# B&R Automation Studio project baseProject
Automation Studio 6.3.1.32; technology packages: mappCockpit 6.2.1, mappMotion 6.3.1, mappSafety 6.2.0, mappServices 6.3.3, mappView 6.3.1, OpcUaCs 6.0.0

## Configuration Config1

CPU X20CP1684, AutomationRuntime 6.0.2, Build 11.3.0, Vc 6.0.0

### Task classes (Cpu.sw)
```
Cyclic#4 (cycle 16000 us, tolerance 16000 us):
  HMI <- HMI.prg
  Safety <- Safety.prg
  motion <- motion.prg
  mappIO <- mappIO.prg
  mappAlarmX <- mappAlarmX.prg
  mappRecipe <- mappRecipe.prg
  EventLog <- EventLog.prg
  Robot <- Robot.prg
Libraries: AsIOAcc, runtime, AsZip, FileIO, astime, sys_lib, ArEventLog, AsBrStr, CoTrace, SfDomain, DataObj, AsMem, AsArProf, standard, MpAlarmX, MpBase, MpAxis, McBase, MpSequence, MpAudit, MpRecipe, MpUserX, MpReport, MpSkyline, MpFile, MpPackML, MpCodeBox, MpCom, MpIO, McAxis, McAcpAx, MpServer
```

### Hardware
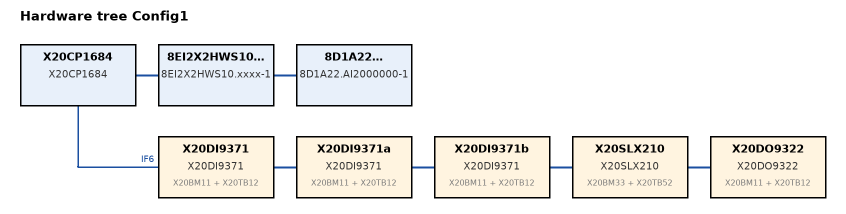
```
8D1A22.AI2000000-1 : 8D1A22.AI2000000-1 v1.0.1.0 (NodeNumber=2)  [PLK1 -> 8EI2X2HWS10.xxxx-1.PLK2 [Cable Type=PowerlinkCable, Length=10, Version=1.0.0.3]]
8EI2X2HWS10.xxxx-1 : 8EI2X2HWS10.xxxx-1 v2.4.0.0 (NodeNumber=1)  [PLK1 -> X20CP1684.IF3 [Cable Type=PowerlinkCable, Length=10, Version=1.0.0.3]; PLK2 -> 8D1A22.AI2000000-1.PLK1 [Cable Type=PowerlinkCable, Length=10, Version=1.0.0.3]]
  DriveConfiguration/Module:
    McAcoposTypeID = AcoposP3SConfig
    ActivateACOPOSSimulationOnPLC = 1
    PowerSupply = AC
  DriveConfiguration/Encoder/EncoderX41:
    InterfaceType = NotUsed
  DriveConfiguration/Channel[1]/RealAxis:
    AxisReference = gAxis_1
    MechanicalElementsIsInvisible = 0
  DriveConfiguration/Channel[1]/RealAxis/MechanicalElements/Gearbox:
    InputIsReadOnly = 0
    Input = 1
    OutputIsReadOnly = 0
    Output = 1
  DriveConfiguration/Channel[1]/RealAxis/MechanicalElements/RotaryToLinearTransformation:
    ReferenceDistanceIsReadOnly = 0
    ReferenceDistance = 1
  DriveConfiguration/Channel[1]/RealAxis:
    EncoderLink = OneEncoder
  DriveConfiguration/Channel[1]/RealAxis/Controller:
    ModeIsReadOnly = 0
    Mode = PositionController
  DriveConfiguration/Channel[1]/RealAxis/Homing:
    ModeIsReadOnly = 0
    Mode = Direct
    RestorePositionVariable = 
  DriveConfiguration/Channel[1]/RealAxis/StopReaction:
    QuickstopIsReadOnly = 0
    Quickstop = DecelerationLimit
    DriveErrorIsReadOnly = 0
    DriveError = DecelerationLimit
  DriveConfiguration/Channel[1]/RealAxis/MovementErrorLimits:
    PositionError = 10.0
    VelocityErrorMonitoring = Automatic1
  DriveConfiguration/Channel[1]/RealAxis:
    JerkFilterIsReadOnly = 0
    JerkFilter = NotUsed
    ZeroVibrationFilter = NotUsed
  DriveConfiguration/Channel[1]/RealAxis/DigitalInputs/HomingSwitch:
    SourceIsReadOnly = 0
    Source = NotUsed
    Level = High
  DriveConfiguration/Channel[1]/RealAxis/DigitalInputs/PositiveLimitSwitch:
    SourceIsReadOnly = 0
    Source = NotUsed
    Level = High
  DriveConfiguration/Channel[1]/RealAxis/DigitalInputs/NegativeLimitSwitch:
    SourceIsReadOnly = 0
    Source = NotUsed
    Level = High
  DriveConfiguration/Channel[1]/RealAxis/DigitalInputs/Trigger1:
    Source = X8Trigger1
    Level = High
  DriveConfiguration/Channel[1]/RealAxis/DigitalInputs/Trigger2:
    Source = X8Trigger2
    Level = High
  DriveConfiguration/Channel[1]/RealAxis/DigitalInputs/Quickstop:
    Input = Trigger2
  DriveConfiguration/Channel[1]/RealAxis/Simulation:
    SimulationModeOnPLC = SetValueGeneration
    SimulationModeOnACOPOS = NotUsed
  DriveConfiguration/Channel[1]:
    VirtualAxis = NotUsed
    ExternalEncoderAxis = NotUsed
X20BM11 : X20BM11 v1.1.0.0  [X2X1 -> X20CP1684.IF6]
X20BM11a : X20BM11 v1.1.0.0  [X2X1 -> X20BM11b.X2X2]
X20BM11b : X20BM11 v1.1.0.0  [X2X1 -> X20BM11.X2X2]
X20BM11c : X20BM11 v1.1.0.0  [X2X1 -> X20BM33.X2X2]
X20BM33 : X20BM33 v1.1.0.0  [X2X1 -> X20BM11a.X2X2]
X20CP1684 : X20CP1684 v1.8.1.0
  Connector IF2:
    ActivateDevice = 1
    Mode = Manual
    InternetAddress = 192.168.50.160
    SubnetMask = 255.255.255.0
  Connector IF3:
    CycleTime = 800
  ConfigurationID = mappView_Config1
  Simulation = 1
  TimerDeviceType = EPLX2X
  TimerDevice = X20CP1684.IF3
  IdleTaskClass = 8
  TaskClassIdleTime = 1600
  Cyclic1Duration = 800
  Cyclic1Tolerance = 0
  Cyclic2Duration = 1600
  Cyclic2Tolerance = 1600
  Cyclic3Duration = 6400
  Cyclic3Tolerance = 6400
  Cyclic4Duration = 16000
  Cyclic4Tolerance = 16000
  Cyclic8Duration = 9600
  FileDevice1
  FileDeviceName1 = USER
  FileDevicePath1 = USER_PATH
  FileDevice2
  FileDeviceName2 = CF
  FileDevicePath2 = C:\
  ActivateFtpServer = 1
  FTPProtocol = 1
  FtpUser1
  FtpUsername1 = ged
  FtpUserPassword1 = mhumPqqez6h0Xcak9Se1xIrLnNOPX6JLQ7ADh5QSq84=
  FtpUserSalt1 = ifft5IbT
  FTPAccessRight1 = 0
  ActivateWebServer = 1
  ActivateSdm = 1
X20DI9371 : X20DI9371 v1.6.1.0  [SS1 -> X20TB12.SS; SL -> X20BM11.SL1]
  Supervision = off
X20DI9371a : X20DI9371 v1.6.1.0  [SS1 -> X20TB12b.SS; SL -> X20BM11b.SL1]
  Supervision = off
X20DI9371b : X20DI9371 v1.6.1.0  [SS1 -> X20TB12a.SS; SL -> X20BM11a.SL1]
  Supervision = off
X20DO9322 : X20DO9322 v1.7.0.0  [SS1 -> X20TB12c.SS; SL -> X20BM11c.SL1]
  Supervision = off
X20SLX210 : X20SLX210 v2.6.1.0  [SS1 -> X20TB52.SS; SL -> X20BM33.SL1]
  Supervision = off
X20TB12 : X20TB12 v1.0.0.0
X20TB12a : X20TB12 v1.0.0.0
X20TB12b : X20TB12 v1.0.0.0
X20TB12c : X20TB12 v1.0.0.0
X20TB52 : X20TB52 v1.0.0.2
```

### IoMap.iom - X20CP1684/IoMap.iom
```iecst
VAR_CONFIG
	::doTestOutput01 AT %QX."X20DO9322".DigitalOutput01;
	::diTestInput01 AT %IX."X20DI9371".DigitalInput01;
	::diTestInput02 AT %IX."X20DI9371a".DigitalInput01;
END_VAR
```

### Config_1.axis - X20CP1684/mappMotion/Config_1.axis
```
Element gAxis_1 (Type=axis)
  BaseType = RotaryPeriodic
  MovementLimits = Internal
  Alarms = None
```

- Safety project (password-protected, skipped)

### Config_2.mpio - X20CP1684/mappServices/Config_2.mpio
```
Element gIoConfig (Type=mpio)
  mapp.Gen:
    Enable = TRUE
    EnableCockpit = TRUE
    Audit = TRUE
    Parent
  Import:
    Main = no
    ImportAllow
    AutoRestore = TRUE
    PreservePv = TRUE
    RemoveLinks = FALSE
    BackupLoc = USER
    TemplateLoc = USER
    Plausibility:
      AllowNarrow = FALSE
      CheckTypes = TRUE
      CheckPv = TRUE
      CheckAxPv = TRUE
  IoDatapoints:
    Inputs:
      0 = #global
    Outputs:
      0 = #global
  Alarms = MpAlarmX
    mapp.AlarmX.Core.Configuration:
      [0]:
        Name = ImportFailed
        Message = {$BR/mapp/MpIO/Alarms/ImportFailed}
        Code = 0
        Severity = 1
        Behavior = EdgeAlarm
          AutoReset = TRUE
          Acknowledge = 1
          Confirm = 0
          MultipleInstances = TRUE
          ReactionWhilePending = TRUE
          Async = FALSE
          Recording:
            InactiveToActive = TRUE
            ActiveToInactive = FALSE
            UnacknowledgedToAcknowledged = TRUE
            UnconfirmedToConfirmed = TRUE
        Disable = FALSE
        AdditionalInformation1
        AdditionalInformation2
      [1]:
        Name = ImportDone
        Message = {$BR/mapp/MpIO/Alarms/ImportDone}
        Code = 0
        Severity = 1
        Behavior = EdgeAlarm
          AutoReset = TRUE
          Acknowledge = 1
          Confirm = 0
          MultipleInstances = TRUE
          ReactionWhilePending = TRUE
          Async = FALSE
          Recording:
            InactiveToActive = TRUE
            ActiveToInactive = FALSE
            UnacknowledgedToAcknowledged = TRUE
            UnconfirmedToConfirmed = TRUE
        Disable = FALSE
        AdditionalInformation1
        AdditionalInformation2
      [2]:
        Name = HwChanged
        Message = {$BR/mapp/MpIO/Alarms/HwChanged}
        Code = 0
        Severity = 1
        Behavior = EdgeAlarm
          AutoReset = TRUE
          Acknowledge = 1
          Confirm = 0
          MultipleInstances = TRUE
          ReactionWhilePending = TRUE
          Async = FALSE
          Recording:
            InactiveToActive = TRUE
            ActiveToInactive = FALSE
            UnacknowledgedToAcknowledged = TRUE
            UnconfirmedToConfirmed = TRUE
        Disable = FALSE
        AdditionalInformation1
        AdditionalInformation2
```

### Config_4.mpalarmxlist - X20CP1684/mappServices/Config_4.mpalarmxlist
```
Element gAlarmXList (Type=mpalarmxlist)
  mapp.AlarmX.Core.Configuration:
    [0]:
      Name = TemperatureHigh
      Message = The Temperature is Too High
      Code = 100
      Severity = 10
      Behavior = PersistentAlarm
        Confirm = 0
        ReactionWhilePending = TRUE
        Retain = FALSE
        Async = FALSE
        DataUpdate:
          Activation:
            TimeStamp = FALSE
            Snippets = FALSE
        Recording:
          InactiveToActive = TRUE
          UnacknowledgedToAcknowledged = TRUE
          AcknowledgedToUnacknowledged = FALSE
          UnconfirmedToConfirmed = TRUE
          ConfirmedToUnconfirmed = FALSE
          Update = FALSE
      Disable = FALSE
      InhibitPV
      AdditionalInformation1
      AdditionalInformation2
  mapp.AlarmX.Snippets:
    AutoDetect = 1
      Language
```

### Config_7.mpfilemanager - X20CP1684/mappServices/Config_7.mpfilemanager
```
Element FileManagement (Type=mpfilemanager)
  mapp.Gen:
    Enable = TRUE
    EnableCockpit = TRUE
    Audit = TRUE
    Parent
  FileManager:
    USB = 1
    Devices:
      0:
        DeviceName = USER
        Text = User
    Access:
      0:
        Folder = *
        Roles:
          0:
            Role = Everyone
            Rights:
              Visible = TRUE
              FolderRead = TRUE
              FileRead = TRUE
              FileEdit = TRUE
              FolderEdit = TRUE
```

## Configuration mappDemoDefault

CPU X20CP1686X, AutomationRuntime 6.0.2, Build 11.3.0, Vc 

### Task classes (Cpu.sw)
```
Cyclic#1:
  MainContro <- MainControl.prg
  ConveyorSi <- ConveyorSim.prg
  Alarm <- Infrastructure.Alarm.prg
Cyclic#4:
  Recipe <- Infrastructure.Recipe.prg
  File <- Infrastructure.File.prg
  Audit <- Infrastructure.Audit.prg
  Report <- Infrastructure.Report.prg
  IO <- Infrastructure.IO.prg
  Sequence <- Infrastructure.Sequence.prg
  CodeBox <- Infrastructure.CodeBox.prg
  PackML <- Industry.PackML.prg
Cyclic#8:
  Skyline <- Infrastructure.Skyline.prg
Binaries: mvLoader, arsvcreg, TCLang, FWRules, udbdef, TCData, mvConfig, CfgFileUI, arconfig, UaCsConfig, CfgFile, mCoWebSc, CfgSkyline, User, TC, asfw, CfgAudit, iomap, Role, CfgReportF, CfgUserX, ashwd, CfgRecipe, CfgSeq, CfgReport, CfgComUnit, ashwac, sysconf, CfgCodeCor, Settings, CfgCodeBox, CfgIO, CfgPack, CfgAlaList, CfgAlaHist, CfgAlaCore, BRRole, CfgHistory, UaDvConfig, CfgAlarm
Libraries: Runtime, Operator, AsIecCon, astime, AsArSdm, DataObj, FileIO, AsBrStr, sys_lib, brsystem, AsArProf, AsMem, standard, AsBrWStr, ArTextSys, ArCert, ArSsl, AsETH, AsHW, AsIOMMan, AsUSB, AsZip, ArUser, UaCoal, UaCoalPrv, ArProject, AsARCfg, CoTrace, MpAlarmX, MpBase, MpSequence, MpAudit, MpRecipe, MpUserX, MpReport, MpSkyline, MpFile, MpPackML, MpCodeBox, MpCom, MpIO, MpServer
```

### Hardware
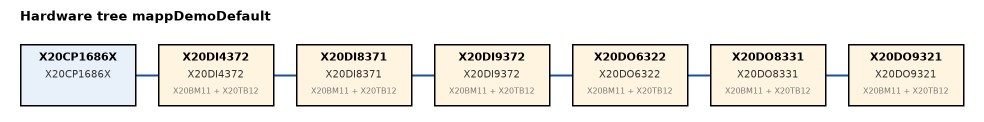
```
X20BM11 : X20BM11 v1.1.0.0  [X2X1 -> X20CP1686X.IF6]
X20BM11a : X20BM11 v1.1.0.0  [X2X1 -> X20BM11.X2X2]
X20BM11b : X20BM11 v1.1.0.0  [X2X1 -> X20BM11a.X2X2]
X20BM11c : X20BM11 v1.1.0.0  [X2X1 -> X20BM11b.X2X2]
X20BM11d : X20BM11 v1.1.0.0  [X2X1 -> X20BM11c.X2X2]
X20BM11e : X20BM11 v1.1.0.0  [X2X1 -> X20BM11d.X2X2]
X20CP1686X : X20CP1686X v1.8.2.0
  Connector IF2:
    ActivateDevice = 1
  ConfigurationID = mappServicesHighlights_Config1
  AutomaticTransferOfUserfiles = on
  Simulation = 1
  FileDevice1
  FileDeviceName1 = HD
  FileDevicePath1 = USER_PATH
  FileDevice2
  FileDeviceName2 = mappDir
  FileDevicePath2 = USER_PATH\mappDemo
  FileDevice3
  FileDeviceName3 = mappReport
  FileDevicePath3 = USER_PATH\mappDemo\Reports
  FileDevice4
  FileDeviceName4 = mappIO
  FileDevicePath4 = USER_PATH\IO
  FileDevice5
  FileDeviceName5 = mappIOBackup
  FileDevicePath5 = USER_PATH\IO\Backup
  FileDevice6
  FileDeviceName6 = mappSequence
  FileDevicePath6 = USER_PATH\Sequence
  FileDevice7
  FileDeviceName7 = mappCodeBox
  FileDevicePath7 = USER_PATH\CodeBox
  ActivateWebServer = 1
  WebServerProtocol = 1
  ActivateSdm = 1
X20DI4372 : X20DI4372 v1.4.1.0  [SS1 -> X20TB12.SS; SL -> X20BM11.SL1]
X20DI8371 : X20DI8371 v1.6.1.0  [SS1 -> X20TB12a.SS; SL -> X20BM11a.SL1]
X20DI9372 : X20DI9372 v1.6.1.0  [SS1 -> X20TB12b.SS; SL -> X20BM11b.SL1]
X20DO6322 : X20DO6322 v1.4.1.0  [SS1 -> X20TB12c.SS; SL -> X20BM11c.SL1]
X20DO8331 : X20DO8331 v1.2.2.0  [SS1 -> X20TB12d.SS; SL -> X20BM11d.SL1]
X20DO9321 : X20DO9321 v1.2.2.0  [SS1 -> X20TB12e.SS; SL -> X20BM11e.SL1]
X20TB12 : X20TB12 v1.0.0.0
X20TB12a : X20TB12 v1.0.0.0
X20TB12b : X20TB12 v1.0.0.0
X20TB12c : X20TB12 v1.0.0.0
X20TB12d : X20TB12 v1.0.0.0
X20TB12e : X20TB12 v1.0.0.0
```

### BRRole.brrole - X20CP1686X/AccessAndSecurity/UserRoleSystem/BRRole.brrole
```
Element BR_Anonymous (Type=BRRole)
Element BR_Engineer (Type=BRRole)
Element BR_Observer (Type=BRRole)
Element BR_SafetyAdmin (Type=BRRole)
Element BR_SecurityAdmin (Type=BRRole)
```

### CfgAlaCore.mpalarmxcore - X20CP1686X/mappServices/CfgAlaCore.mpalarmxcore
```
Element gAlarmXCore (Type=mpalarmxcore)
  mapp.Gen:
    Enable = TRUE
    TaskClass = 4
  mapp.AlarmX.List:
    [0]:
      List = gAlarmXCore_List
      Offset = 0
  mapp.AlarmX.Create = Disabled
  mapp.AlarmX.Core.Retain:
    Memory = 0
```

### CfgAlaHist.mpalarmxhistory - X20CP1686X/mappServices/CfgAlaHist.mpalarmxhistory
```
Element gAlarmXHistory (Type=mpalarmxhistory)
  mapp.Gen:
    Audit = TRUE
  mapp.AlarmX.History
```

### CfgAlaList.mpalarmxlist - X20CP1686X/mappServices/CfgAlaList.mpalarmxlist
```
Element gAlarmXCore_List (Type=mpalarmxlist)
  mapp.AlarmX.Core.Configuration:
    [0]:
      Name = RecordingStarted
      Message = {$mappDemo/MpDataUserAlarm}
      Code = 2501
      Behavior = UserDefined
        AutoReset = TRUE
        Acknowledge = 0
        Recording:
          ActiveToInactive = FALSE
    [1]:
      Name = WaterEmpty
      Message = {$IAT/AlarmWater}
      Code = 2503
      Behavior = LevelMonitoring
        Monitoring:
          MonitoredPV = ::MainContro:Refill[3]
          LowLimitEnable = Static
            Limit = 15
      AdditionalInformation1 = WaterEmpty
    [2]:
      Name = CoffeeEmpty
      Message = {$IAT/AlarmCoffee}
      Code = 2504
      Behavior = LevelMonitoring
        Monitoring:
          MonitoredPV = ::MainContro:Refill[0]
          LowLimitEnable = Static
            Limit = 15
      AdditionalInformation1 = CoffeeEmpty
    [3]:
      Name = MilkEmpty
      Message = {$IAT/AlarmMilk}
      Code = 2505
      Behavior = LevelMonitoring
        Monitoring:
          MonitoredPV = ::MainContro:Refill[1]
          LowLimitEnable = Static
            Limit = 15
      AdditionalInformation1 = MilkEmpty
    [4]:
      Name = SugarEmpty
      Message = {$IAT/AlarmSugar}
      Code = 2506
      Behavior = LevelMonitoring
        Monitoring:
          MonitoredPV = ::MainContro:Refill[2]
          LowLimitEnable = Static
            Limit = 15
      AdditionalInformation1 = SugarEmpty
    [5]:
      Name = ModuleAlarm
      Message = {$IAT/AlarmModule}
      Behavior = PersistentAlarm
  mapp.AlarmX.Snippets:
    [0]:
      Key = WaterLevel
      Value:
        PV = ::MainContro:Refill[3]
    [1]:
      Key = SugarLevel
      Value:
        PV = ::MainContro:Refill[2]
    [2]:
      Key = CoffeeLevel
      Value:
        PV = ::MainContro:Refill[0]
    [3]:
      Key = MilkLevel
      Value:
        PV = ::MainContro:Refill[1]
```

### CfgAudit.mpaudittrail - X20CP1686X/mappServices/CfgAudit.mpaudittrail
```
Element gAuditTrail (Type=mpaudittrail)
  mapp.Gen:
    Enable = TRUE
    TaskClass = 8
  Audit:
    Events:
      [0] = 600
      [1] = 400
      [2] = 1000
      [3] = 1001
      [4] = 1002
      [5] = 1003
      [6] = 700
      [7] = 701
      [8] = 702
      [9] = 703
      [10] = 704
      [11] = 100
      [12] = 101
      [13] = 102
      [14] = 103
      [15] = 104
      [16] = 105
      [17] = 106
      [18] = 107
      [19] = 108
      [20] = 150
      [21] = 151
      [22] = 152
      [23] = 153
      [24] = 154
      [25] = 155
      [26] = 156
      [27] = 157
      [28] = 158
      [29] = 159
      [30] = 160
      [31] = 161
      [32] = 162
      [33] = 163
      [34] = 164
      [35] = 165
      [36] = 166
      [37] = 167
      [38] = 168
      [39] = 169
      [40] = 170
      [41] = 171
      [42] = 300
      [43] = 301
      [44] = 302
      [45] = 303
      [46] = 350
      [47] = 351
      [48] = 352
      [49] = 353
    RecordMemory = 1
    RecordingSize = 200
    SramBufferSize = 4
    TextSource:
      DisplayFormat = {$AuditDisplay/Root}
      ExportFormat = {$AuditExport/Root}
    Archive = On
      Mode = 0
      Time = 0
      MaxSize = 100
    Export:
      RawData = FALSE
      FileType = 0
      Encrypt = FALSE
      PassPhrase = Insert your passphrase here...
  Monitor:
    0:
      pv = ::Recipe:CoffeeIngredients.Milk
      id = Milk
    1:
      pv = ::Recipe:CoffeeIngredients.Water
      id = Water
    2:
      pv = ::Recipe:CoffeeIngredients.Sugar
      id = Sugar
    3:
      pv = ::Recipe:CoffeeIngredients.Coffee
      id = Coffee
  Alarms = MpAlarmX
    mapp.AlarmX.Core.Configuration:
      [0]:
        Name = ArchiveAvailable
        Message = {$BR/mapp/MpAuditTrail/Alarms/ArchiveAvailable}
        Code = 0
        Severity = 1
        Behavior = PersistentAlarm
          AutoReset = FALSE
          Acknowledge = 1
          Confirm = 0
          MultipleInstances = FALSE
          ReactionWhilePending = TRUE
          Async = FALSE
          DataUpdate:
            Activation:
              TimeStamp = FALSE
              Snippets = FALSE
          Recording:
            InactiveToActive = TRUE
            ActiveToInactive = FALSE
            UnacknowledgedToAcknowledged = TRUE
            AcknowledgedToUnacknowledged = TRUE
            UnconfirmedToConfirmed = TRUE
            ConfirmedToUnconfirmed = TRUE
            Update = FALSE
        Disable = FALSE
        AdditionalInformation1
        AdditionalInformation2
      [1]:
        Name = MaxArchives
        Message = {$BR/mapp/MpAuditTrail/Alarms/MaxArchives}
        Code = 0
        Severity = 1
        Behavior = EdgeAlarm
          AutoReset = TRUE
          Acknowledge = 1
          Confirm = 0
          MultipleInstances = TRUE
          ReactionWhilePending = TRUE
          Async = FALSE
          Recording:
            InactiveToActive = TRUE
            ActiveToInactive = FALSE
            UnacknowledgedToAcknowledged = TRUE
            UnconfirmedToConfirmed = TRUE
        Disable = FALSE
        AdditionalInformation1
        AdditionalInformation2
```

### CfgComUnit.mpcomunit - X20CP1686X/mappServices/CfgComUnit.mpcomunit
```
Element gGroup (Type=mpcomunit)
  Display:
    Groups:
      0:
        Id = Fluid
        DisplayUnits:
          Metric:
            Code = MLT
          Imperial:
            Code = OZA
          ImperialUS:
            Code = OZA
      1:
        Id = Gram
        DisplayUnits:
          Metric:
            Code = GRM
          Imperial:
            Code = ONZ
          ImperialUS:
            Code = ONZ
    Datapoints:
      0:
        Id = ::Recipe:CoffeeIngredients.Milk
        DisplayUnits = UnitGroup
          Unitgroup = Fluid
      1:
        Id = ::Recipe:CoffeeIngredients.Water
        DisplayUnits = UnitGroup
          Unitgroup = Fluid
      2:
        Id = ::Recipe:CoffeeIngredients.Sugar
        DisplayUnits = UnitGroup
          Unitgroup = Gram
      3:
        Id = ::Recipe:CoffeeIngredients.Coffee
        DisplayUnits = UnitGroup
          Unitgroup = Gram
      4:
        Id = ::MainContro:Refill[1]
        DisplayUnits = UnitGroup
          Unitgroup = Fluid
      5:
        Id = ::MainContro:Refill[2]
        DisplayUnits = UnitGroup
          Unitgroup = Gram
      6:
        Id = ::MainContro:Refill[0]
        DisplayUnits = UnitGroup
          Unitgroup = Gram
      7:
        Id = ::MainContro:Refill[3]
        DisplayUnits = UnitGroup
          Unitgroup = Fluid
    Units:
      0:
        EngineeringUnit:
          Code = MLT
        DisplayUnits:
          Metric:
            Code = MLT
          Imperial:
            Code = MLT
          ImperialUS:
            Code = MLT
      1:
        EngineeringUnit:
          Code = MLT
        DisplayUnits:
          Metric:
            Code = MLT
          Imperial:
            Code = MLT
          ImperialUS:
            Code = MLT
      2:
        EngineeringUnit:
          Code = GRM
        DisplayUnits:
          Metric:
            Code = GRM
          Imperial:
            Code = ONZ
          ImperialUS:
            Code = ONZ
      3:
        EngineeringUnit:
          Code = GRM
        DisplayUnits:
          Metric:
            Code = GRM
          Imperial:
            Code = ONZ
          ImperialUS:
            Code = ONZ
```

### CfgFile.mpfilemanager - X20CP1686X/mappServices/CfgFile.mpfilemanager
```
Element FileManagement (Type=mpfilemanager)
  mapp.Gen:
    Enable = TRUE
    EnableCockpit = TRUE
    Audit = TRUE
    Parent
  FileManager:
    USB = 0
    Devices:
      0:
        DeviceName = mappDir
        Text = Recipe files
    Access:
      0:
        Folder = *
        Roles:
          0:
            Role = Everyone
            Rights:
              Visible = TRUE
              FolderRead = TRUE
              FileRead = TRUE
              FileEdit = TRUE
              FolderEdit = TRUE
          1:
            Role = Administrators
            Rights:
              Visible = TRUE
              FolderRead = TRUE
              FileRead = TRUE
              FileEdit = TRUE
              FolderEdit = TRUE
  FileManagerRestrict:
    0:
      Functionality = TextEditor
```

### CfgPack.mppackmlstandaloneunit - X20CP1686X/mappServices/CfgPack.mppackmlstandaloneunit
```
Element gPackMLStandaloneUnit (Type=mppackmlstandaloneunit)
  mapp.Gen:
    Enable = TRUE
    TaskClass = 1
    Audit = TRUE
  Settings:
    StartupActiveMode = 1
    WarningStateTransNotAllowed = FALSE
    WarningModeTransNotAllowed = FALSE
    ModeActivationCmdLevel = FALSE
    StartupActiveState = 4
    PackTags = 0
  Modes:
    Mode[1]:
      ModeID = 1
      Name = Production
      State[0] = 0
      State[1] = 0
      State[2] = 1
        AllowIn = TRUE
        AllowOut = TRUE
      State[3] = 1
        AllowIn = FALSE
        AllowOut = FALSE
      State[4] = 1
        AllowIn = TRUE
        AllowOut = TRUE
      State[5] = 0
      State[6] = 1
        AllowIn = FALSE
        AllowOut = FALSE
      State[7] = 1
        AllowIn = FALSE
        AllowOut = FALSE
      State[8] = 1
        AllowIn = FALSE
        AllowOut = FALSE
      State[9] = 1
        AllowIn = TRUE
        AllowOut = TRUE
      State[10] = 0
      State[11] = 0
      State[12] = 0
      State[13] = 0
      State[14] = 0
      State[15] = 1
        AllowIn = FALSE
        AllowOut = FALSE
      State[16] = 1
        AllowIn = FALSE
        AllowOut = FALSE
      State[17] = 0
```

### CfgRecipe.mprecipexml - X20CP1686X/mappServices/CfgRecipe.mprecipexml
```
Element gRecipeXml (Type=mprecipexml)
  mapp.Gen:
    Enable = TRUE
    TaskClass = 4
    Audit = TRUE
  mapp.Recipe.Xml:
    AutoSave = Standard
    Encryption = FALSE
    PassPhrase = 
    AutoExtension = TRUE
    Signature = Disabled
  Alarms = MpAlarmX
    mapp.AlarmX.Core.Configuration:
      [0]:
        Name = SaveFailed
        Message = {$BR/mapp/MpRecipeXml/Alarms/SaveFailed}
        Code = 0
        Severity = 1
        Behavior = EdgeAlarm
          AutoReset = TRUE
          Acknowledge = 1
          Confirm = 0
          MultipleInstances = TRUE
          ReactionWhilePending = TRUE
          Async = FALSE
          Recording:
            InactiveToActive = TRUE
            ActiveToInactive = FALSE
            UnacknowledgedToAcknowledged = TRUE
            UnconfirmedToConfirmed = TRUE
        Disable = FALSE
        AdditionalInformation1
        AdditionalInformation2
      [1]:
        Name = SaveFailedPartial
        Message = {$BR/mapp/MpRecipeXml/Alarms/SaveFailedPartial}
        Code = 0
        Severity = 1
        Behavior = EdgeAlarm
          AutoReset = TRUE
          Acknowledge = 1
          Confirm = 0
          MultipleInstances = TRUE
          ReactionWhilePending = TRUE
          Async = FALSE
          Recording:
            InactiveToActive = TRUE
            ActiveToInactive = FALSE
            UnacknowledgedToAcknowledged = TRUE
            UnconfirmedToConfirmed = TRUE
        Disable = FALSE
        AdditionalInformation1
        AdditionalInformation2
      [2]:
        Name = LoadFailed
        Message = {$BR/mapp/MpRecipeXml/Alarms/LoadFailed}
        Code = 0
        Severity = 1
        Behavior = EdgeAlarm
          AutoReset = TRUE
          Acknowledge = 1
          Confirm = 0
          MultipleInstances = TRUE
          ReactionWhilePending = TRUE
          Async = FALSE
          Recording:
            InactiveToActive = TRUE
            ActiveToInactive = FALSE
            UnacknowledgedToAcknowledged = TRUE
            UnconfirmedToConfirmed = TRUE
        Disable = FALSE
        AdditionalInformation1
        AdditionalInformation2
      [3]:
        Name = LoadFailedPartial
        Message = {$BR/mapp/MpRecipeXml/Alarms/LoadFailedPartial}
        Code = 0
        Severity = 1
        Behavior = EdgeAlarm
          AutoReset = TRUE
          Acknowledge = 1
          Confirm = 0
          MultipleInstances = TRUE
          ReactionWhilePending = TRUE
          Async = FALSE
          Recording:
            InactiveToActive = TRUE
            ActiveToInactive = FALSE
            UnacknowledgedToAcknowledged = TRUE
            UnconfirmedToConfirmed = TRUE
        Disable = FALSE
        AdditionalInformation1
        AdditionalInformation2
```

### CfgReport.mpreportcore - X20CP1686X/mappServices/CfgReport.mpreportcore
```
Element gReport (Type=mpreportcore)
  mapp.Gen:
    Enable = TRUE
    EnableCockpit = TRUE
    Parent
  MpReport:
    Settings:
      ResourceDeviceName = HD
      LanguageDependent:
        [0]:
          Language = de
          Font = 1
          DateTimePattern = %Y-%m-%d %H:%M:%S
          PrecisionDateTimePattern = %Y-%m-%d %H:%M:%S,%L
        [1]:
          Language = en
          Font = 1
          DateTimePattern = %Y-%m-%d %H:%M:%S
          PrecisionDateTimePattern = %Y-%m-%d %H:%M:%S,%L
    PageLayouts:
      [0]:
        Name = Default
        PageFormat = 4
        Orientation = 1
        Margins = 1
    Styles:
      Text:
        [0]:
          Name = Default
          Style = 0
          Size = 12
          Color = 000000
          Precision = 6
        [1]:
          Name = Header
          Style = 1
          Size = 20
          Color = FF9900
          Precision = 6
        [2]:
          Name = Subheader
          Style = 0
          Size = 16
          Color = FF9900
          Precision = 6
      Table:
        [0]:
          Name = Default
          BorderWidth = 1
          Color = 000000
          Padding = 10
          HeadRowOnNewPage = FALSE
      Line:
        [0]:
          Name = Default
          Width = 1
          Color = FF9900
      Chart:
        PieChart:
          [0]:
            Name = Default
            BackColor = FFFFFF
            BorderWidth = 0
            BorderColor = 000000
            Padding = 1
            ItemBorderWidth = 0
            ItemBorderColor = 000000
        LineChart:
          [0]:
            Name
            BackColor = FFFFFF
            BorderWidth = 1
            BorderColor = 000000
            Padding = 1
            GraphBackColor = FFFFFF
            GraphBorderWidth = 1
            GraphBorderColor = 000000
            GridLineWidth = 1
            GridLineColor = 000000
        BarChart:
          [0]:
            Name
            BackColor = FFFFFF
            BorderWidth = 1
            BorderColor = 000000
            Padding = 1
            ItemGapWidth = 1
            GraphBackColor = FFFFFF
            GraphBorderWidth = 1
            GraphBorderColor = 000000
            GridLineWidth = 1
            GridLineColor = 000000
    Tables:
      [0] = ColumnsByRow
        Name = CoffeeInformation
        TableStyle = Default
        TextStyle = Default
        [0]:
          MinimumHeight = 10
          [0] = TextId
            Source = {$Report/ReportData}
            Width = 50
            HorizontalAlign = 0
            TextStyleReference = InheritedTextStyle
          [1] = TextId
            Source = {$Report/ReportValue}
            Width = 50
            HorizontalAlign = 0
            TextStyleReference = InheritedTextStyle
        [1]:
          MinimumHeight = 10
          [0] = TextId
            Source = {$Report/ReportCurrCoffee}
            Width = 50
            HorizontalAlign = 0
            TextStyleReference = InheritedTextStyle
          [1] = ValueId
            Value = ProcessVariable
              ProcessVariable = ::Recipe:LoadRecipeSimple
              UnitDisplay = 0
            Width = 50
            HorizontalAlign = 0
            TextStyleReference = InheritedTextStyle
        [2]:
          MinimumHeight = 10
          [0] = TextId
            Source = {$Report/ReportMilk}
            Width = 50
            HorizontalAlign = 0
            TextStyleReference = InheritedTextStyle
          [1] = ValueId
            Value = ProcessVariable
              ProcessVariable = ::Recipe:CoffeeIngredients.Milk
              UnitDisplay = 1
            Width = 50
            HorizontalAlign = 0
            TextStyleReference = InheritedTextStyle
        [3]:
          MinimumHeight = 10
          [0] = TextId
            Source = {$Report/ReportWater}
            Width = 50
            HorizontalAlign = 0
            TextStyleReference = InheritedTextStyle
          [1] = ValueId
            Value = ProcessVariable
              ProcessVariable = ::Recipe:CoffeeIngredients.Water
              UnitDisplay = 1
            Width = 50
            HorizontalAlign = 0
            TextStyleReference = InheritedTextStyle
        [4]:
          MinimumHeight = 10
          [0] = TextId
            Source = {$Report/ReportSugar}
            Width = 50
            HorizontalAlign = 0
            TextStyleReference = InheritedTextStyle
          [1] = ValueId
            Value = ProcessVariable
              ProcessVariable = ::Recipe:CoffeeIngredients.Sugar
              UnitDisplay = 1
            Width = 50
            HorizontalAlign = 0
            TextStyleReference = InheritedTextStyle
        [5]:
          MinimumHeight = 10
          [0] = TextId
            Source = {$Report/ReportCoffee}
            Width = 50
            HorizontalAlign = 0
            TextStyleReference = InheritedTextStyle
          [1] = ValueId
            Value = ProcessVariable
              ProcessVariable = ::Recipe:CoffeeIngredients.Coffee
              UnitDisplay = 1
            Width = 50
            HorizontalAlign = 0
            TextStyleReference = InheritedTextStyle
    Contents:
      [0]:
        Name = Discription
        [0] = Text
          Text = {$Report/ReportDescription}
          HorizontalAlign = 0
          NewLine = TRUE
          TextStyle = Default
      [1]:
        Name = Table
        [0] = Table
          Table = CoffeeInformation
          HorizontalAlign = 1
      [2]:
        Name = Underline
        [0] = Line
          LineStyle = Default
      [3]:
        Name = Header
        [0] = Text
          Text = {$Report/ReportHeader}
          HorizontalAlign = 1
          NewLine = TRUE
          TextStyle = Header
      [4]:
        Name = EmptyLine
        [0] = EmptyLine
          Size = 10
    Reports:
      [0]:
        Name = ReportCoffee
        Settings:
          OwnerPassword
          UserPassword
          AllowPrint = TRUE
          AllowCopy = FALSE
          AllowEdit = FALSE
        PageLayout = Default
        Header = Header
        Footer
        [0]:
          StartOnNewPage = FALSE
          Heading:
            Text
            HorizontalAlign = 0
            TextStyle
          [0]:
            Content = Underline
            Width = 100
        [1]:
          StartOnNewPage = FALSE
          Heading:
            Text
            HorizontalAlign = 0
            TextStyle
          [0]:
            Content = EmptyLine
            Width = 100
        [2]:
          StartOnNewPage = FALSE
          Heading:
            Text = {$Report/ReportDescriptionHeader}
            HorizontalAlign = 0
            TextStyle = Subheader
          [0]:
            Content = Discription
            Width = 100
        [3]:
          StartOnNewPage = FALSE
          Heading:
            Text
            HorizontalAlign = 0
            TextStyle
          [0]:
            Content = EmptyLine
            Width = 100
        [4]:
          StartOnNewPage = FALSE
          Heading:
            Text = {$Report/ReportHeaderTable}
            HorizontalAlign = 0
            TextStyle = Subheader
          [0]:
            Content = Table
            Width = 100
        [5]:
          StartOnNewPage = FALSE
          Heading:
            Text
            HorizontalAlign = 0
            TextStyle
          [0]:
            Content = EmptyLine
            Width = 100
  Alarms = MpAlarmX
    mapp.AlarmX.Core.Configuration:
      [0]:
        Name = GenerateFailed
        Message = {$BR/mapp/MpReportCore/Alarms/GenerateFailed}
        Code = 0
        Severity = 1
        Behavior = EdgeAlarm
          AutoReset = TRUE
          Acknowledge = 1
          Confirm = 0
          MultipleInstances = TRUE
          ReactionWhilePending = TRUE
          Async = FALSE
          Recording:
            InactiveToActive = TRUE
            ActiveToInactive = FALSE
            UnacknowledgedToAcknowledged = TRUE
            UnconfirmedToConfirmed = TRUE
        Disable = FALSE
        AdditionalInformation1
        AdditionalInformation2
```

### CfgSkyline.mpskyline - X20CP1686X/mappServices/CfgSkyline.mpskyline
```
Element gSkyline (Type=mpskyline)
  MpSkyline:
    ModuleStateCollections:
      [0]:
        Name = CoffeeMachineStates
        States:
          [0]
          [1]:
            Name = Ready
          [2]:
            Name = Warning
          [3]:
            Name = Error
    OptionStateCollections:
      [0]:
        Name = CoolingStates
        States:
          [0]:
            Name = Off
          [1]:
            Name = Cooling
      [1]:
        Name = HeatingStates
        States:
          [0]:
            Name = Off
          [1]:
            Name = Heating
      [2]:
        Name = FilterStates
        States:
          [0]:
            Name = NormalFilter
          [1]:
            Name = PremiumFilter
      [3]:
        Name = GrinderStates
        States:
          [0]:
            Name = GrindRough
          [1]:
            Name = GrindFine
    NotificationCollections:
      [0]:
        Name = CoffeeNotifications
        Notifications:
          [0]:
            Name = Information
          [1]:
            Name = Alarm
    Options:
      [0]:
        Name = OptionCooling
        OptionStateCollection = CoolingStates
      [1]:
        Name = OptionHeating
        OptionStateCollection = HeatingStates
      [2]:
        Name = OptionFilter
        OptionStateCollection = FilterStates
      [3]:
        Name = OptionGrinder
        OptionStateCollection = GrinderStates
    ModuleTypes:
      [0]:
        Name = Unit_Tank
        Size = L
        StateCollection = CoffeeMachineStates
        NotificationCollection = CoffeeNotifications
        [0]:
          Name = OptionCooling
        [1]:
          Name = OptionHeating
      [1]:
        Name = Unit_Filter
        Size = L
        StateCollection = CoffeeMachineStates
        NotificationCollection = CoffeeNotifications
        [0]:
          Name = OptionFilter
      [2]:
        Name = Unit_Grinder
        Size = M
        StateCollection = CoffeeMachineStates
        NotificationCollection = CoffeeNotifications
        [0]:
          Name = OptionGrinder
      [3]:
        Name = Unit_Start
        Size = M
        StateCollection = CoffeeMachineStates
        NotificationCollection = CoffeeNotifications
      [4]:
        Name = Unit_End
        Size = L
        StateCollection = CoffeeMachineStates
        NotificationCollection = CoffeeNotifications
    Modules:
      [0]:
        Name = Start
        Type = Unit_Start
        Grouping = 0
      [1]:
        Name = Water_Tank
        Type = Unit_Tank
      [2]:
        Name = Coffee_Tank
        Type = Unit_Tank
      [3]:
        Name = Milk_Tank
        Type = Unit_Tank
      [4]:
        Name = Filtering
        Type = Unit_Filter
        Grouping = 0
      [5]:
        Name = Sugar_Tank
        Type = Unit_Tank
      [6]:
        Name = Coffee_Grinder
        Type = Unit_Grinder
        Grouping = 0
      [7]:
        Name = End
        Type = Unit_End
        Grouping = 0
```

### CfgUserX.mpuserx - X20CP1686X/mappServices/CfgUserX.mpuserx
```
Element UserMgmtX (Type=mpuserx)
  mapp.Gen:
    Audit = TRUE
  UserMgmtSystem:
    UserMgmtSystemType = 0
  ServerSettings:
    Server = ADServer
      Timeout = 10
      Mapping:
        TableName
      DisplayName = Username
  PasswordPolicy:
    PasswordMaxAge = 0
    PasswordExpirationNotification = 0
    PasswordHistory = 0
    PasswordChangeReq = FALSE
    PasswordCase = FALSE
    PasswordAlpha = FALSE
    PasswordSpecial = FALSE
    PasswordLength = 3
  UserAccount:
    InvalidPasswordAttempts = 3
    UserExpirationTime = 0
    AutoLogoutTime = 3600
    UserNameLength = 1
    NoDelete = FALSE
    AdminUnlockTime = 3600
    EditSameLevel = 1
  ImportExport:
    ImportUser = 2
    ImportRole = 2
    ImportUnchecked = FALSE
  Users:
    DefUser#1:
      id = admin
      name = Admin
      lang = en
      measSystem = 1
    DefUser#2:
      id = Anonymous
      name
      lang
      measSystem = 0
  Roles:
    DefRole#1:
      id = Administrators
      level = 100
      admin = TRUE
    DefRole#2:
      id = Everyone
      level = 10
      admin = FALSE
    DefRole#3:
      id = BR_Engineer
      level = 100
      admin = TRUE
    DefRole#4:
      id = BR_SecurityAdmin
      level = 120
      admin = TRUE
```

## Logical view

Binary libraries used (declarations not repeated): operator, runtime, AsIecCon, astime, AsIOAcc, AsZip, FileIO, sys_lib, ArEventLog, AsBrStr, AsArSdm, DataObj, brsystem, AsArProf, AsMem, standard, AsBrWStr, ArTextSys, ArCert, ArSsl, ArUser, AsETH, AsHW, AsIOMMan, AsUSB, CoTrace, SfDomain 6.2.0, MpAlarmX 6.3.3, MpBase, MpAxis 6.3.1, McBase 6.3.1, MpSequence 6.3.3, MpAudit 6.3.3, MpRecipe 6.3.3, MpUserX 6.3.3, MpReport 6.3.3, MpSkyline 6.3.3, MpFile 6.3.3, MpPackML 6.3.3, MpCodeBox 6.3.3, MpCom 6.3.3, MpIO 6.3.3, McAxis 6.3.1, McAcpAx 6.3.1, MpServer

### Global.typ - Global data types
```iecst
TYPE
	Machine_Settings_typ : 	STRUCT
		CO_Width : REAL;
		CO_Width_Preset_Val : REAL; (*Cutoff Width Display Preset Value*)
		Life_Crimps : UDINT;
		Crimp_Time : UINT;
		crimpTime : TIME;
		PE_Offset : REAL;
		PE_Offset_Raw : REAL;
		Cutoff_Length : REAL; (*Cutoff Length*)
		Cutoff_Length_Finish : REAL; (*Cutoff Finish Length*)
		Corner_Punch_Count : UDINT; (*Number of Corner Punches*)
		Life_Corner_Punch_Count : UDINT; (*Number of Corner Punches, Lifetime*)
		Cut_Count : UDINT; (*Number of Cutoff Punches*)
		Life_Cut_Count : UDINT; (*Number of Cutoff Punches, Lifetime*)
		Gag_Cyl_Count : UDINT; (*Number of Gag Cylinder Actuations*)
		Life_Gag_Cyl_Count : UDINT; (*Number of Gag Cylinder Actuations, Lifetime*)
		Hole_Punch_Count : UDINT; (*Number of Registration Hole Punches*)
		Life_Hole_Punch_Count : UDINT; (*Number of Registration Hole Punches, Lifetime*)
		End_Start_Punch_Count : UDINT; (*Number of End Start Punches*)
		Life_End_Start_Punch_Count : UDINT; (*Number of End Start Punches, Lifetime*)
		Shear_Punch_Count : UDINT; (*Number of Shear Punches*)
		Life_Shear_Punch_Count : UDINT; (*Number of Shear Punches, Lifetime*)
		Muntin_Punch_Count : UDINT; (*Number of Muntin Punches*)
		Life_Muntin_Punch_Count : UDINT; (*Number of Miter Punches, Lifetime*)
		Tab_Punch_Count : UDINT; (*Number of Tab Punches*)
		Life_Tab_Punch_Count : UDINT; (*Number of Tab Punches, Lifetime*)
		Dimple_Punch_Count : UDINT; (*Number of Dimple Punches*)
		Life_Dimple_Punch_Count : UDINT; (*Number of Dimple Punches, Lifetime*)
		Material_Length : REAL; (*Length of Material that has been run through Feeder Press*)
		Life_Material_Length : REAL; (*Length of Material that has been run through Feeder Press, Lifetime*)
		Scrap_Max_Length : REAL;
		Max_Length : REAL;
		Last_Unit_Distance : DINT;
		First_Unit_Distance : DINT;
		FP_Width : REAL;
		FP_Width_Preset_Val : REAL; (*Feeder Press Width Display Preset Value*)
		RF_Width : REAL;
		RF_Width_Preset_Val : REAL; (*Rollformer Width Display Preset Value*)
		HMI_2_QC_Pos : BOOL;
		HMI_2_TP1 : BOOL;
		HMI_2_TP2 : BOOL;
		HMI_2_UL1 : BOOL;
		HMI_2_UL2 : BOOL;
		HMI_2_BL1 : BOOL;
		HMI_2_BL2 : BOOL;
		HMI_2_UB1 : BOOL;
		HMI_2_UB2 : BOOL;
		Conveyor_Speed : USINT;
		System_Drift_Disable : BOOL; (*Disable All Drift Shutdowns*)
		HomeOffset : ARRAY[0..7]OF REAL;
		CrimpDelay : DINT;
		CrimperEnable : BOOL;
		FeederPressExtractionTime : UINT;
		FeederPressFeedLength : REAL;
		CrimperPEOffset : REAL;
		RollformerClearDistance : REAL;
		RollformerThreadUpDistance : REAL;
		LightCurtainDisable : BOOL;
		ExtruderDisable : BOOL;
	END_STRUCT;
	PackMLModes :
		(
		PACKML_MODE_PRODUCTION := 1,
		PACKML_MODE_MAINTENANCE := 2
		);
	ReportCoffeeType : 	STRUCT
		Name : STRING[255];
		Water : INT;
		Sugar : INT;
		Coffee : INT;
		Milk : INT;
	END_STRUCT;
	RefillAlarmType : 	STRUCT
		Water : INT;
		Sugar : INT;
		Milk : INT;
		Coffee : INT;
	END_STRUCT;
	RefillType : 	STRUCT
		Water : INT;
		Sugar : INT;
		Milk : INT;
		Coffee : INT;
	END_STRUCT;
	CoffeeMainLogicType : 	STRUCT  (*Main logic structure *)
		AxisCupFeeder : CoffeeAxisLogicType; (*Control structure for axis*)
		AxisTakeout : CoffeeAxisLogicType; (*Control structure for axis*)
		cmdAbort : BOOL; (*HMI control to start the brewing process*)
		cmdStop : BOOL; (*HMI control to start the brewing process*)
		cmdClear : BOOL; (*HMI control to start the brewing process*)
		cmdStart : BOOL; (*HMI control to start the brewing process*)
		TemperatureWithinLimit : BOOL; (*HMI control bit *)
		CreateFirstRecipe : BOOL; (*Enable synchronization when creating the default recipes*)
		cmdTakeout : BOOL;
		Refill : ARRAY[0..3]OF INT; (*Structure to control the ingredients*)
		AlarmRefill : ARRAY[0..3]OF INT; (*Structure which is controlling the Refill-Alarms*)
		CoffeeState : CoffeeStateEnum;
		ReportCoffee : ARRAY[0..199]OF ReportCoffeeType;
		PackMLState : STRING[80];
		IdleState : BOOL;
	END_STRUCT;
	CoffeeAxisLogicType : 	STRUCT  (*Sub structure for controlling axis*)
		Active : BOOL; (*Axis component is ready*)
		Power : BOOL; (*Power on command*)
		PowerOn : BOOL; (*Power is on*)
		Home : BOOL; (*Homing command *)
		MoveAdditive : BOOL; (*MoveAdditive command*)
		MoveActive : BOOL; (*Move active*)
		InPosition : BOOL; (*Commanded position reached *)
		Position : LREAL; (*Current position*)
	END_STRUCT;
	CoffeeStateEnum :
		(
		COFFEE_WAIT := 0,
		COFFEE_TAKEWATER := 1,
		COFFEE_TAKECOFFEE := 2,
		COFFEE_TAKECOFFEEMILK := 3,
		COFFEE_RELEASE := 4,
		COFFEE_FINISH := 5
		);
END_TYPE
```

### Global.var - Global variables
```iecst
VAR
	doTestOutput01 : BOOL;
	diTestInput02 : BOOL;
	diTestInput01 : BOOL;
END_VAR
VAR RETAIN
	Machine_Settings : Machine_Settings_typ; (*Machine Parameters that are Remanent*)
END_VAR
(*Definitions for main components of the coffee machine*)
VAR
	gUnit : STRING[80] := 'metric'; (*Get unit from visualization*)
	gSetUnit : INT := 1; (*Set the current unit*)
	gClearAlarm : BOOL := FALSE; (*Check if Alarm can be cleared*)
	gCoffeeMainLogic : CoffeeMainLogicType; (*Control structure of main logic*)
	gSetLanguage : STRING[80] := 'en'; (*Set the current language*)
END_VAR
```

### Package Logical/Libraries - Global libraries

- Visualisation Logical/mappView (not shown)

### Program Logical/HMI (IEC)

#### Variables.var
```iecst
VAR
	speed : INT;
	temperature : REAL;
	start : BOOL;
	ArEventLogCreate_0 : ArEventLogCreate;
END_VAR
```

#### Main.st
```iecst
PROGRAM _INIT
	(* Insert code here *)

END_PROGRAM

PROGRAM _CYCLIC
	//mappView HMI test, Automation Studio 6.0

	speed;
	temperature;
	start;

END_PROGRAM

PROGRAM _EXIT
	(* Insert code here *)

END_PROGRAM
```

### Program Logical/Safety (IEC)

#### Types.typ
```iecst
TYPE
	StepEnum :
		(
		WAIT,
		CONNECT,
		TRANSFER,
		COMP_READ_INFO,
		COMP_WAIT_ACK,
		COMPLETION,
		DISCONNECT
		);
END_TYPE
```

#### Variables.var
```iecst
VAR
	SfDomainCompletion_0 : SfDomainCompletion;
	SfDomainInfo_0 : SfDomainInfo;
	SfDomainTransfer_0 : SfDomainTransfer;
	SfDomainConnect_0 : SfDomainConnect;
	Step : StepEnum;
	bCmdStart : BOOL;
	bDataCorrect : BOOL;
	Station : STRING[80];
	AsIOAccRead_0 : AsIOAccRead;
	bootState : UDINT;
END_VAR
```

#### Main.st
```iecst
PROGRAM _INIT
   (* SfDomainConnect *)
	SfDomainConnect_0.SfDomain := ADR(gSafeDomain_1);
	(* Username and password defined under UserRoleSystem in the Configuration View *)
	SfDomainConnect_0.UserName := 'ged';
	SfDomainConnect_0.Password := 'ged';

	(* SfDomainTransfer *)
	SfDomainTransfer_0.SfDomain := ADR(gSafeDomain_1);
	(* Name of the SafeAPPLICATION and SafeCOMMISSIONING to be transferred *)
	SfDomainTransfer_0.SafeAppFilePath := 'mapp1.sfapp';
	SfDomainTransfer_0.SafeCommFilePath := '';

	(* SfDomainInfo *)
	SfDomainInfo_0.SfDomain := ADR(gSafeDomain_1);

	(* SfDomainCompletion *)
	SfDomainCompletion_0.SfDomain := ADR(gSafeDomain_1);

END_PROGRAM

PROGRAM _CYCLIC

	CASE Step OF

		(* Wait for the command to start machine commissioning *)
		WAIT:
			IF bCmdStart THEN
				Step := CONNECT;
			END_IF

			(* Establish connection to the SafeDOMAIN *)
		CONNECT:
			SfDomainConnect_0.Enable := TRUE;
			IF SfDomainConnect_0.Active = TRUE THEN
				Step := TRANSFER;
			END_IF

			(* Transfer the SafeAPPLICATION and SafeCOMMISSIONING to the SafeDOMAIN *)
		TRANSFER:
			SfDomainTransfer_0.Execute := TRUE;
			IF SfDomainTransfer_0.Done = TRUE THEN
				SfDomainTransfer_0.Execute := FALSE;
				Step := COMP_READ_INFO;
			END_IF

			(* Read information from the SafeDOMAIN *)
		COMP_READ_INFO:
			SfDomainInfo_0.Execute := TRUE;
			IF SfDomainInfo_0.Done = TRUE THEN
				SfDomainInfo_0.Execute := FALSE;
				(* Copy the read information to function block SfDomainCompletion, *)
				(* display this data for verification *)
				SfDomainCompletion_0.Info := SfDomainInfo_0.Info;
				Step := COMP_WAIT_ACK;
			END_IF

			(* Wait for acknowledgment *)
			(* User acknowledges correctness with bDataCorrect = TRUE *)
		COMP_WAIT_ACK:
			IF bDataCorrect THEN
				bDataCorrect := FALSE;
				Step := COMPLETION;
			END_IF

			(* Finish step completion *)
		COMPLETION:
			SfDomainCompletion_0.Execute := TRUE;
			IF SfDomainCompletion_0.Done = TRUE THEN
				SfDomainCompletion_0.Execute := FALSE;
				Step := DISCONNECT;
			END_IF

			(* Disconnect from the SafeDOMAIN *)
		DISCONNECT:
			SfDomainConnect_0.Enable := FALSE;
			IF SfDomainConnect_0.Busy = FALSE THEN
				bCmdStart := FALSE;
				Step := WAIT;
			END_IF

	END_CASE

	Station := 'IF6.ST4';
	AsIOAccRead_0(enable := TRUE, pDeviceName := ADR(Station), pChannelName := ADR('SLXbootState'));		//Added 3/21/18

	IF AsIOAccRead_0.status = 0 THEN
		bootState := AsIOAccRead_0.value;
	ELSIF AsIOAccRead_0.status <> 65535 THEN
		bootState := 0;
	END_IF

	(* Cyclic call of the function blocks *)
	SfDomainConnect_0();
	SfDomainTransfer_0();
	SfDomainInfo_0();
	SfDomainCompletion_0();

END_PROGRAM

PROGRAM _EXIT
	(* Insert code here *)

END_PROGRAM
```

### Program Logical/mappIO (IEC)

#### Variables.var
```iecst
VAR
	MpIOImport_0 : MpIOImport;
	configTemplateName : STRING[80];
END_VAR
```

#### Main.st
```iecst
PROGRAM _INIT
	configTemplateName := 'NewConfig';

END_PROGRAM

PROGRAM _CYCLIC

	MpIOImport_0.MpLink := ADR(gIoConfig);
	MpIOImport_0.Enable := TRUE;
	MpIOImport_0.FileName := ADR(configTemplateName);
	MpIOImport_0.DeviceName := ADR('USER');

	MpIOImport_0();

	//test IO points
	diTestInput01;
	diTestInput02;

	doTestOutput01;

END_PROGRAM

PROGRAM _EXIT
	(* Insert code here *)

END_PROGRAM
```

### Program Logical/mappAlarmX (IEC)

#### Variables.var
```iecst
VAR
	MpAlarmXCore_0 : MpAlarmXCore;
	MpAlarmXHistory_0 : MpAlarmXHistory;
	Temperature : INT;
END_VAR
```

#### Main.st
```iecst
PROGRAM _INIT
	MpAlarmXCore_0.Enable := TRUE;
	MpAlarmXCore_0.MpLink := ADR(gAlarmXCore);

	MpAlarmXHistory_0.Enable := TRUE;
	MpAlarmXHistory_0.MpLink := ADR(gAlarmXHistory);
	MpAlarmXHistory_0.FileName := ADR('Alarms_%Y_%m_%d_%H_%M_%S');
	//MpAlarmXHistory_0.DeviceName := ADR('CF');
	MpAlarmXHistory_0.DeviceName := ADR('USER');

	MpAlarmXCore_0();
	MpAlarmXHistory_0();

END_PROGRAM

PROGRAM _CYCLIC

	IF Temperature >= 50 THEN
		MpAlarmXSet(gAlarmXCore,'TemperatureHigh');
	ELSE
		MpAlarmXReset(gAlarmXCore,'TemperatureHigh');
	END_IF;

	MpAlarmXCore_0();
	MpAlarmXHistory_0();

END_PROGRAM

PROGRAM _EXIT

END_PROGRAM
```

### Program Logical/mappRecipe (IEC)

#### Variables.var
```iecst
VAR
	MpRecipeRegPar_0 : MpRecipeRegPar;
	MpRecipeXML_0 : MpRecipeXml;
	recipeXML : INT;
	loadSettings : BOOL;
	saveSettings : BOOL;
END_VAR
```

#### Main.st
```iecst
PROGRAM _INIT
	(* Insert code here *)

END_PROGRAM

PROGRAM _CYCLIC
	Machine_Settings.Hole_Punch_Count;
	Machine_Settings.Last_Unit_Distance;
	Machine_Settings.Life_Corner_Punch_Count;
	Machine_Settings.Life_Crimps;
	Machine_Settings.Life_Cut_Count;
	Machine_Settings.Life_Dimple_Punch_Count;
	Machine_Settings.Life_Gag_Cyl_Count;
	Machine_Settings.Life_Hole_Punch_Count;
	Machine_Settings.Life_Material_Length;
	Machine_Settings.Life_Muntin_Punch_Count;
	Machine_Settings.Life_Tab_Punch_Count;
	Machine_Settings.Material_Length;
	Machine_Settings.Max_Length;
	Machine_Settings.Muntin_Punch_Count;
	Machine_Settings.PE_Offset;
	Machine_Settings.PE_Offset_Raw;

	//mapp recipe stuff

	CASE recipeXML OF
		0:
			IF loadSettings = TRUE THEN
				recipeXML := 10;
			END_IF
			IF saveSettings = TRUE THEN
				recipeXML := 30;
			END_IF

		10:	//load
			MpRecipeXML_0.Load := TRUE;
			recipeXML := 20;

		20:
			IF MpRecipeXML_0.CommandDone = TRUE THEN
				loadSettings := FALSE;
				MpRecipeXML_0.Load := FALSE;
				recipeXML := 0;
			END_IF

		30:	//save
			MpRecipeXML_0.Save := TRUE;
			recipeXML := 40;

		40:
			IF MpRecipeXML_0.CommandDone = TRUE THEN
				saveSettings := FALSE;
				MpRecipeXML_0.Save := FALSE;
				recipeXML := 0;
			END_IF

	END_CASE

	//Function block calls
	MpRecipeXML_0(MpLink := ADR(gRecipeXml), Enable := TRUE, DeviceName := ADR('USER'), FileName := ADR('MachineSettings'));
	MpRecipeRegPar_0(MpLink := ADR(gRecipeXml) , Enable := TRUE, PVName := ADR('Machine_Settings'));

END_PROGRAM

PROGRAM _EXIT
	(* Insert code here *)

END_PROGRAM
```

### Program Logical/EventLog (IEC)

#### EventLog.st
```iecst
(********************************************************************
 * COPYRIGHT -- Bernecker + Rainer
 ********************************************************************
 * PROGRAM: EventLog
 * File: EventLog.st
 * Author: Bernecker + Rainer
 * Created: June, 2015
 ********************************************************************
 * Implementation OF PROGRAM EventLog
 ********************************************************************)

PROGRAM _INIT
	EventLog.Event.EnteredBy := 'UserID';
	brsstrcpy(ADR(EventLog.Event.AdditionalData), ADR('This is an information entry from the user.'));
	EventLog.Event.AdditionalDataSize := brsstrlen(ADR(EventLog.Event.AdditionalData)) + 1;
	EventLog.Event.AdditionalDataFormat := arEVENTLOG_ADDFORMAT_TEXT;
	(*See ArEventLog help for the description of the event id, facilities 0-15 are reserved for customer use.*)
	EventLog.Event.EventID := ArEventLogMakeEventID(Severity := arEVENTLOG_SEVERITY_INFO, Facility := 10, ErrorCode := 1024);
END_PROGRAM

PROGRAM _CYCLIC
	CASE EventLog.Data.Step OF
		(*Waits for user input (command).*)
		STEP_WAIT_FOR_INPUT:
			IF EventLog.Commands.CreateUserLog THEN
				EventLog.Commands.CreateUserLog := FALSE;
				EventLog.Data.Step := STEP_GET_LOGBOOK_IDENT;
				EventLog.Data.GetIdentFailNextStep := STEP_CREATE_LOGBOOK;
				EventLog.Data.GetIdentOkNextStep := STEP_WAIT_FOR_INPUT;
			ELSIF EventLog.Commands.DeleteUserLog THEN
				EventLog.Commands.DeleteUserLog := FALSE;
				EventLog.Data.Step := STEP_GET_LOGBOOK_IDENT;
				EventLog.Data.GetIdentFailNextStep := STEP_ERROR;
				EventLog.Data.GetIdentOkNextStep := STEP_DELETE_LOGBOOK;
			ELSIF EventLog.Commands.WriteUserEvent THEN
				EventLog.Commands.WriteUserEvent := FALSE;
				EventLog.Data.Step := STEP_GET_LOGBOOK_IDENT;
				EventLog.Data.GetIdentFailNextStep := STEP_ERROR;
				EventLog.Data.GetIdentOkNextStep := STEP_WRITE_EVENT;
			ELSIF EventLog.Commands.ReadLatestEvent THEN
				EventLog.Commands.ReadLatestEvent := FALSE;
				EventLog.Data.Step := STEP_GET_LOGBOOK_IDENT;
				EventLog.Data.GetIdentFailNextStep := STEP_ERROR;
				EventLog.Data.GetIdentOkNextStep := STEP_GET_LATEST_RECORD_ID;
			ELSIF EventLog.Commands.ReadPreviousEvent THEN
				EventLog.Commands.ReadPreviousEvent := FALSE;
				EventLog.Data.Step := STEP_GET_LOGBOOK_IDENT;
				EventLog.Data.GetIdentFailNextStep := STEP_ERROR;
				EventLog.Data.GetIdentOkNextStep := STEP_GET_PREVIOUS_RECORD_ID;
			END_IF

		(*Gets the ident of the user logbook "UsrEvLog".*)
		STEP_GET_LOGBOOK_IDENT:
			IF EventLog.FunctionBlocks.ArEventLogGetIdent_0.Done THEN
				EventLog.FunctionBlocks.ArEventLogGetIdent_0.Execute := FALSE;
				EventLog.Data.Ident := EventLog.FunctionBlocks.ArEventLogGetIdent_0.Ident;
				EventLog.Data.StatusID := ERR_OK;
				EventLog.Data.Step := EventLog.Data.GetIdentOkNextStep;
			ELSIF EventLog.FunctionBlocks.ArEventLogGetIdent_0.Error THEN
				EventLog.FunctionBlocks.ArEventLogGetIdent_0.Execute := FALSE;
				EventLog.Data.StatusID := EventLog.FunctionBlocks.ArEventLogGetIdent_0.StatusID;
				EventLog.Data.Step := EventLog.Data.GetIdentFailNextStep;
			ELSE
				(*Execute the FB only if the ident isn't already set.*)
				IF EventLog.Data.Ident = 0 THEN
					EventLog.FunctionBlocks.ArEventLogGetIdent_0.Name := 'UsrEvLog';
					EventLog.FunctionBlocks.ArEventLogGetIdent_0.Execute := TRUE;
				ELSE
					EventLog.Data.StatusID := ERR_OK;
					EventLog.Data.Step := EventLog.Data.GetIdentOkNextStep;
				END_IF
			END_IF

		(*Creates the user logbook "UsrEvLog".*)
		STEP_CREATE_LOGBOOK:
			IF EventLog.FunctionBlocks.ArEventLogCreate_0.Done THEN
				EventLog.FunctionBlocks.ArEventLogCreate_0.Execute := FALSE;
				EventLog.Data.Ident := EventLog.FunctionBlocks.ArEventLogCreate_0.Ident;
				EventLog.Data.StatusID := ERR_OK;
				EventLog.Data.Step := STEP_WAIT_FOR_INPUT;
			ELSIF EventLog.FunctionBlocks.ArEventLogCreate_0.Error THEN
				EventLog.FunctionBlocks.ArEventLogCreate_0.Execute := FALSE;
				EventLog.Data.StatusID := EventLog.FunctionBlocks.ArEventLogCreate_0.StatusID;
				EventLog.Data.Step := STEP_ERROR;
			ELSE
				EventLog.FunctionBlocks.ArEventLogCreate_0.Name := 'UsrEvLog';
				EventLog.FunctionBlocks.ArEventLogCreate_0.Size := 10000;
				EventLog.FunctionBlocks.ArEventLogCreate_0.Persistence := arEVENTLOG_PERSISTENCE_PERSIST;
				EventLog.FunctionBlocks.ArEventLogCreate_0.Info := 0;
				EventLog.FunctionBlocks.ArEventLogCreate_0.Execute := TRUE;
			END_IF

		(*Deletes the user logbook "UsrEvLog".*)
		STEP_DELETE_LOGBOOK:
			IF EventLog.FunctionBlocks.ArEventLogDelete_0.Done THEN
				EventLog.FunctionBlocks.ArEventLogDelete_0.Execute := FALSE;
				EventLog.Data.Ident := 0;
				EventLog.Data.StatusID := ERR_OK;
				EventLog.Data.Step := STEP_WAIT_FOR_INPUT;
			ELSIF EventLog.FunctionBlocks.ArEventLogDelete_0.Error THEN
				EventLog.FunctionBlocks.ArEventLogDelete_0.Execute := FALSE;
				EventLog.Data.StatusID := EventLog.FunctionBlocks.ArEventLogDelete_0.StatusID;
				EventLog.Data.Step := STEP_ERROR;
			ELSE
				EventLog.FunctionBlocks.ArEventLogDelete_0.Ident := EventLog.Data.Ident;
				EventLog.FunctionBlocks.ArEventLogDelete_0.Execute := TRUE;
			END_IF

		(*Writes the event set in EventLog.Event to the user logbook "UsrEvLog".*)
		STEP_WRITE_EVENT:
			IF EventLog.FunctionBlocks.ArEventLogWrite_0.Done THEN
				EventLog.FunctionBlocks.ArEventLogWrite_0.Execute := FALSE;
				EventLog.Data.StatusID := ERR_OK;
				EventLog.Data.Step := STEP_WAIT_FOR_INPUT;
			ELSIF EventLog.FunctionBlocks.ArEventLogWrite_0.Error THEN
				EventLog.FunctionBlocks.ArEventLogWrite_0.Execute := FALSE;
				EventLog.Data.StatusID := EventLog.FunctionBlocks.ArEventLogWrite_0.StatusID;
				EventLog.Data.Step := STEP_ERROR;
			ELSE
				EventLog.FunctionBlocks.ArEventLogWrite_0.Ident := EventLog.Data.Ident;
				EventLog.FunctionBlocks.ArEventLogWrite_0.EventID := EventLog.Event.EventID;
				EventLog.FunctionBlocks.ArEventLogWrite_0.TimeStamp := 0; (*System timestamp.*)
				EventLog.FunctionBlocks.ArEventLogWrite_0.ObjectID := EventLog.Event.EnteredBy;
				EventLog.FunctionBlocks.ArEventLogWrite_0.OriginRecordID := EventLog.Event.OriginID;
				EventLog.FunctionBlocks.ArEventLogWrite_0.AddDataFormat := EventLog.Event.AdditionalDataFormat;
				EventLog.FunctionBlocks.ArEventLogWrite_0.AddDataSize := EventLog.Event.AdditionalDataSize;
				EventLog.FunctionBlocks.ArEventLogWrite_0.AddData := ADR(EventLog.Event.AdditionalData);
				EventLog.FunctionBlocks.ArEventLogWrite_0.Execute := TRUE;
			END_IF

		(*Gets the id of the latest record in the user logbook "UsrEvLog".*)
		STEP_GET_LATEST_RECORD_ID:
			IF EventLog.FunctionBlocks.ArEventLogGetLatestRecordID_0.Done THEN
				EventLog.FunctionBlocks.ArEventLogGetLatestRecordID_0.Execute := FALSE;
				EventLog.Event.RecordID := EventLog.FunctionBlocks.ArEventLogGetLatestRecordID_0.RecordID;
				EventLog.Data.StatusID := ERR_OK;
				EventLog.Data.Step := STEP_READ_EVENT;
			ELSIF EventLog.FunctionBlocks.ArEventLogGetLatestRecordID_0.Error THEN
				EventLog.FunctionBlocks.ArEventLogGetLatestRecordID_0.Execute := FALSE;
				EventLog.Data.StatusID := EventLog.FunctionBlocks.ArEventLogGetLatestRecordID_0.StatusID;
				EventLog.Data.Step := STEP_ERROR;
			ELSE
				EventLog.FunctionBlocks.ArEventLogGetLatestRecordID_0.Ident := EventLog.Data.Ident;
				EventLog.FunctionBlocks.ArEventLogGetLatestRecordID_0.Execute := TRUE;
			END_IF

		(*Gets the id of the previous record of the given record id (EventLog.Event.RecordID).*)
		STEP_GET_PREVIOUS_RECORD_ID:
			IF EventLog.FunctionBlocks.ArEventLogGetPreviousRecordID_0.Done THEN
				EventLog.FunctionBlocks.ArEventLogGetPreviousRecordID_0.Execute := FALSE;
				EventLog.Event.RecordID := EventLog.FunctionBlocks.ArEventLogGetPreviousRecordID_0.PrevRecordID;
				EventLog.Data.StatusID := ERR_OK;
				EventLog.Data.Step := STEP_READ_EVENT;
			ELSIF EventLog.FunctionBlocks.ArEventLogGetPreviousRecordID_0.Error THEN
				EventLog.FunctionBlocks.ArEventLogGetPreviousRecordID_0.Execute := FALSE;
				EventLog.Data.StatusID := EventLog.FunctionBlocks.ArEventLogGetPreviousRecordID_0.StatusID;
				EventLog.Data.Step := STEP_ERROR;
			ELSE
				EventLog.FunctionBlocks.ArEventLogGetPreviousRecordID_0.Ident := EventLog.Data.Ident;
				EventLog.FunctionBlocks.ArEventLogGetPreviousRecordID_0.RecordID := EventLog.Event.RecordID;
				EventLog.FunctionBlocks.ArEventLogGetPreviousRecordID_0.Execute := TRUE;
			END_IF

		(*Reads the event with the given record id from the to user logbook "UsrEvLog".*)
		STEP_READ_EVENT:
			IF EventLog.FunctionBlocks.ArEventLogRead_0.Done THEN
				EventLog.FunctionBlocks.ArEventLogRead_0.Execute := FALSE;
				EventLog.Event.AdditionalDataFormat := EventLog.FunctionBlocks.ArEventLogRead_0.AddDataFormat;
				EventLog.Event.AdditionalDataSize := EventLog.FunctionBlocks.ArEventLogRead_0.AddDataSize;
				EventLog.Event.TimeStamp := EventLog.FunctionBlocks.ArEventLogRead_0.TimeStamp;
				EventLog.Event.OriginID := EventLog.FunctionBlocks.ArEventLogRead_0.OriginRecordID;
				EventLog.Data.StatusID := ERR_OK;
				EventLog.Event.ErrorNumber := 0;
				EventLog.Event.Customer := ArEventLogIsCustomerArea(EventID := EventLog.FunctionBlocks.ArEventLogRead_0.EventID);
				EventLog.Event.Severity := GetSeverity(EventID := EventLog.FunctionBlocks.ArEventLogRead_0.EventID);
				EventLog.Event.Code := GetCode(EventID := EventLog.FunctionBlocks.ArEventLogRead_0.EventID);
				EventLog.Event.Facility := GetFacility(EventID := EventLog.FunctionBlocks.ArEventLogRead_0.EventID);
				IF EventLog.FunctionBlocks.ArEventLogRead_0.StatusID = arEVENTLOG_WRN_NO_EVENTID THEN
					(*The given record id is not an event id record. Invoke ArEventLogReadErrorNumber to read the error number and the severity.*)
					EventLog.Data.Step := STEP_READ_ERROR_NUMBER;
				ELSIF EventLog.Event.AdditionalDataSize > 0 THEN
					EventLog.Data.Step := STEP_READ_ADDITIONAL_DATA;
				ELSE
					EventLog.Data.Step := STEP_READ_OBJECT_ID;
				END_IF
			ELSIF EventLog.FunctionBlocks.ArEventLogRead_0.Error THEN
				EventLog.FunctionBlocks.ArEventLogRead_0.Execute := FALSE;
				EventLog.Data.StatusID := EventLog.FunctionBlocks.ArEventLogRead_0.StatusID;
				EventLog.Data.Step := STEP_ERROR;
			ELSE
				EventLog.FunctionBlocks.ArEventLogRead_0.Ident := EventLog.Data.Ident;
				EventLog.FunctionBlocks.ArEventLogRead_0.RecordID := EventLog.Event.RecordID;
				EventLog.FunctionBlocks.ArEventLogRead_0.Execute := TRUE;
			END_IF

		(*Reads the error number event with the given record id from the user logbook "UsrEvLog".*)
		STEP_READ_ERROR_NUMBER:
			IF EventLog.FunctionBlocks.ArEventLogReadErrorNumber_0.Done THEN
				EventLog.FunctionBlocks.ArEventLogReadErrorNumber_0.Execute := FALSE;
				EventLog.Event.ErrorNumber := EventLog.FunctionBlocks.ArEventLogReadErrorNumber_0.ErrorNumber;
				EventLog.Event.Severity := EventLog.FunctionBlocks.ArEventLogReadErrorNumber_0.Severity;
				EventLog.Data.StatusID := ERR_OK;
				IF EventLog.Event.AdditionalDataSize > 0 THEN
					EventLog.Data.Step := STEP_READ_ADDITIONAL_DATA;
				ELSE
					EventLog.Data.Step := STEP_READ_OBJECT_ID;
				END_IF
			ELSIF EventLog.FunctionBlocks.ArEventLogReadErrorNumber_0.Error THEN
				EventLog.FunctionBlocks.ArEventLogReadErrorNumber_0.Execute := FALSE;
				EventLog.Data.StatusID := EventLog.FunctionBlocks.ArEventLogReadErrorNumber_0.StatusID;
				EventLog.Data.Step := STEP_ERROR;
			ELSE
				EventLog.FunctionBlocks.ArEventLogReadErrorNumber_0.Ident := EventLog.Data.Ident;
				EventLog.FunctionBlocks.ArEventLogReadErrorNumber_0.RecordID := EventLog.Event.RecordID;
				EventLog.FunctionBlocks.ArEventLogReadErrorNumber_0.Execute := TRUE;
			END_IF

		(*Reads the additional data of the event with the given record id from the user logbook "UsrEvLog".*)
		STEP_READ_ADDITIONAL_DATA:
			IF EventLog.FunctionBlocks.ArEventLogReadAddData_0.Done THEN
				EventLog.FunctionBlocks.ArEventLogReadAddData_0.Execute := FALSE;
				EventLog.Event.AdditionalDataSize := EventLog.FunctionBlocks.ArEventLogReadAddData_0.AddDataSize;
				EventLog.Data.StatusID := ERR_OK;
				EventLog.Data.Step := STEP_READ_OBJECT_ID;
			ELSIF EventLog.FunctionBlocks.ArEventLogReadAddData_0.Error THEN
				EventLog.FunctionBlocks.ArEventLogReadAddData_0.Execute := FALSE;
				EventLog.Data.StatusID := EventLog.FunctionBlocks.ArEventLogReadAddData_0.StatusID;
				EventLog.Data.Step := STEP_ERROR;
			ELSE
				EventLog.FunctionBlocks.ArEventLogReadAddData_0.Ident := EventLog.Data.Ident;
				EventLog.FunctionBlocks.ArEventLogReadAddData_0.RecordID := EventLog.Event.RecordID;
				EventLog.FunctionBlocks.ArEventLogReadAddData_0.BytesToRead := SIZEOF(EventLog.Event.AdditionalData);
				EventLog.FunctionBlocks.ArEventLogReadAddData_0.AddData := ADR(EventLog.Event.AdditionalData);
				EventLog.FunctionBlocks.ArEventLogReadAddData_0.Execute := TRUE;
			END_IF

		(*Reads the object id of the event with the given record id from the user logbook "UsrEvLog".*)
		STEP_READ_OBJECT_ID:
			IF EventLog.FunctionBlocks.ArEventLogReadObjectID_0.Done THEN
				EventLog.FunctionBlocks.ArEventLogReadObjectID_0.Execute := FALSE;
				EventLog.Event.EnteredBy := EventLog.FunctionBlocks.ArEventLogReadObjectID_0.ObjectID;
				EventLog.Data.StatusID := ERR_OK;
				EventLog.Data.Step := STEP_WAIT_FOR_INPUT;
			ELSIF EventLog.FunctionBlocks.ArEventLogReadObjectID_0.Error THEN
				EventLog.FunctionBlocks.ArEventLogReadObjectID_0.Execute := FALSE;
				EventLog.Data.StatusID := EventLog.FunctionBlocks.ArEventLogReadObjectID_0.StatusID;
				EventLog.Data.Step := STEP_ERROR;
			ELSE
				EventLog.FunctionBlocks.ArEventLogReadObjectID_0.Ident := EventLog.Data.Ident;
				EventLog.FunctionBlocks.ArEventLogReadObjectID_0.RecordID := EventLog.Event.RecordID;
				EventLog.FunctionBlocks.ArEventLogReadObjectID_0.Execute := TRUE;
			END_IF

		STEP_ERROR:
		(*Do some error handling here.*)
	END_CASE

	EventLog.FunctionBlocks.ArEventLogCreate_0;
	EventLog.FunctionBlocks.ArEventLogDelete_0;
	EventLog.FunctionBlocks.ArEventLogWrite_0;
	EventLog.FunctionBlocks.ArEventLogGetIdent_0;
	EventLog.FunctionBlocks.ArEventLogGetLatestRecordID_0;
	EventLog.FunctionBlocks.ArEventLogGetPreviousRecordID_0;
	EventLog.FunctionBlocks.ArEventLogReadAddData_0;
	EventLog.FunctionBlocks.ArEventLogReadErrorNumber_0;
	EventLog.FunctionBlocks.ArEventLogReadObjectID_0;
	EventLog.FunctionBlocks.ArEventLogRead_0;
END_PROGRAM

(*See ArEventLog help for the description of the event id format!*)

(*Gets severity from EventId (bits 31-30).*)
FUNCTION GetSeverity
	IF ArEventLogIsError(EventID := EventID) THEN
		GetSeverity := arEVENTLOG_SEVERITY_ERROR;
	ELSIF ArEventLogIsWarning(EventID := EventID) THEN
		GetSeverity := arEVENTLOG_SEVERITY_WARNING;
	ELSIF ArEventLogIsInformation(EventID := EventID) THEN
		GetSeverity := arEVENTLOG_SEVERITY_INFO;
	ELSIF ArEventLogIsSuccess(EventID := EventID) THEN
		GetSeverity := arEVENTLOG_SEVERITY_SUCCESS;
	END_IF
END_FUNCTION

(*Gets code from EventId (bits 15-0).*)
FUNCTION GetCode
	GetCode := DINT_TO_UINT(EventID);
END_FUNCTION

(*Gets facility from EventId (bits 27-16).*)
FUNCTION GetFacility
	GetFacility := DINT_TO_UINT(SHR(EventID, 16) AND 16#0FFF);
END_FUNCTION
```

#### EventLog.typ
```iecst
(********************************************************************
 * COPYRIGHT -- Bernecker + Rainer
 ********************************************************************
 * Program: EventLog
 * File: EventLog.typ
 * Author: Bernecker + Rainer
 * Created: June, 2015
 ********************************************************************
 * Local data types of program EventLog
 ********************************************************************)

TYPE
	EventLog_typ : 	STRUCT  (*Event handling.*)
		Commands : EventLog_Commands_typ; (*Event handling user commands.*)
		Data : EventLog_Data_typ; (*Event handling data for state machine.*)
		Event : EventLog_Event_typ; (*Event handling event description.*)
		FunctionBlocks : EventLog_FunctionBlocks_typ; (*Event handling used functionblocks.*)
	END_STRUCT;
	EventLog_Commands_typ : 	STRUCT
		CreateUserLog : BOOL; (*Creates the user logbook "UsrEvLog" in USERROM.*)
		DeleteUserLog : BOOL; (*Deletes the user logbook "UsrEvLog".*)
		WriteUserEvent : BOOL; (*Writes a user event into the user logbook "UsrEvLog". *)
		ReadLatestEvent : BOOL; (*Reads the latest event of the user logbook "UsrEvLog".*)
		ReadPreviousEvent : BOOL; (*Reads the previous event (of the given record id) of the user logbook "UserEvLog".*)
	END_STRUCT;
	EventLog_Data_typ : 	STRUCT
		Step : EventLogSteps; (*Current step. STEP_ERROR must be manually reset (STEP_WAIT_FOR_INPUT).*)
		Ident : ArEventLogIdentType; (*Ident of the logbook "UsrEvLog".*)
		StatusID : DINT; (*Status information for STEP_ERROR.*)
		GetIdentOkNextStep : EventLogSteps; (*Internal helper for state machine.*)
		GetIdentFailNextStep : EventLogSteps; (*Internal helper for state machine.*)
	END_STRUCT;
	EventLog_Event_typ : 	STRUCT
		Severity : USINT; (*Severity of the last event (read).*)
		Customer : BOOL; (*Customer bit of the last event (read).*)
		Facility : UINT; (*Facility of the last event (read).*)
		Code : UINT; (*Code of the last event (read).*)
		EventID : DINT; (*EventID for write event (write - is not set by reading an event).*)
		ErrorNumber : UDINT; (*Error number of the event- set when the read event is no event id event (read).*)
		EnteredBy : STRING[36]; (*User/object identification (read/write - optional).*)
		OriginID : ArEventLogRecordIDType; (*Record id of the origin record (read/write - optional).*)
		RecordID : ArEventLogRecordIDType; (*Record id of the event to read (read - set automatically).*)
		TimeStamp : ArEventLogTimeStampType;
		AdditionalDataSize : UDINT; (*Size of the additional data (read/write - optional)*)
		AdditionalDataFormat : USINT; (*Format of the additional data (read/write)*)
		AdditionalData : ARRAY[0..128]OF USINT; (*Additional data (read/write)*)
	END_STRUCT;
	EventLog_FunctionBlocks_typ : 	STRUCT
		ArEventLogCreate_0 : ArEventLogCreate;
		ArEventLogDelete_0 : ArEventLogDelete;
		ArEventLogGetIdent_0 : ArEventLogGetIdent;
		ArEventLogGetLatestRecordID_0 : ArEventLogGetLatestRecordID;
		ArEventLogGetPreviousRecordID_0 : ArEventLogGetPreviousRecordID;
		ArEventLogWrite_0 : ArEventLogWrite;
		ArEventLogRead_0 : ArEventLogRead;
		ArEventLogReadErrorNumber_0 : ArEventLogReadErrorNumber;
		ArEventLogReadAddData_0 : ArEventLogReadAddData;
		ArEventLogReadObjectID_0 : ArEventLogReadObjectID;
	END_STRUCT;
	EventLogSteps :
		(
		STEP_WAIT_FOR_INPUT := 0,
		STEP_CREATE_LOGBOOK := 1,
		STEP_DELETE_LOGBOOK := 2,
		STEP_GET_LOGBOOK_IDENT := 3,
		STEP_WRITE_EVENT := 4,
		STEP_READ_EVENT := 5,
		STEP_READ_ERROR_NUMBER := 6,
		STEP_READ_ADDITIONAL_DATA := 7,
		STEP_READ_OBJECT_ID := 8,
		STEP_GET_LATEST_RECORD_ID := 9,
		STEP_GET_PREVIOUS_RECORD_ID := 10,
		STEP_ERROR := 255
		);
END_TYPE
```

#### EventLog.var
```iecst
(********************************************************************
 * COPYRIGHT -- Bernecker + Rainer
 ********************************************************************
 * Program: EventLog
 * File: EventLog.var
 * Author: Bernecker + Rainer
 * Created: June, 2015
 ********************************************************************
 * Local variables of program EventLog
 ********************************************************************)
VAR
	EventLog : EventLog_typ; (*Event handling.*)
END_VAR
```

#### EventLog.fun
```iecst
FUNCTION GetSeverity : USINT (*Gets severity from EventId (bits 31-30).*)
	VAR_INPUT
		EventID : DINT;
	END_VAR
END_FUNCTION

FUNCTION GetFacility : UINT (*Gets facility from EventId (bits 27-16).*)
	VAR_INPUT
		EventID : DINT;
	END_VAR
END_FUNCTION

FUNCTION GetCode : UINT (*Gets code from EventId (bits 15-0).*)
	VAR_INPUT
		EventID : DINT;
	END_VAR
END_FUNCTION
```

### Program Logical/Robot (IEC)

#### Variables.var
```iecst
VAR
	Sensor2 : BOOL;
	Sensor3 : BOOL;
	Sensor1 : BOOL;
	ConveyorSpeed : REAL;
	ActivateConveyor : BOOL;
	RobotOutput : ARRAY[0..1] OF USINT;
	RobotInput : ARRAY[0..1] OF USINT;
END_VAR
```

#### Main.st
```iecst
PROGRAM _INIT
	(* Insert code here *)

END_PROGRAM

PROGRAM _CYCLIC
//robot variables
	Sensor1;
	Sensor2;
	Sensor3;
	ActivateConveyor;
	ConveyorSpeed;
	RobotInput;
	RobotOutput;

END_PROGRAM

PROGRAM _EXIT
	(* Insert code here *)

END_PROGRAM
```

### Package Logical/Infrastructure - Infrastructure Components

### Program Logical/Infrastructure/Alarm (IEC) - Alarm handling

#### Variables.var
```iecst
VAR
	MpAlarmXHistory_0 : MpAlarmXHistory; (*MpAlarmXHistory instance*)
	MpAlarmXListUI_0 : MpAlarmXListUI; (*MpAlarmXList instance*)
	MpAlarmXCore_0 : MpAlarmXCore; (*MpAlarmXCore instance*)
	ChangeStyleAlarmButton : USINT := 0; (*changeStyle of a AlarmFlyout in mappView*)
	AlarmButton : BOOL := FALSE; (*Contol Variable for Button in mapp View*)
	MpAlarmXListUIConnect : MpAlarmXListUIConnectType := (0);
	AlarmVideo : WSTRING[255] := "";
	AlarmInfo : BOOL := 0;
	FilterConfiguration : STRING[1000] := '';
	SortConfiguration : STRING[1000] := '';
	HistoryFilter : STRING[2000] := '';
	HistorySort : STRING[2000] := '';
	Test : INT := 0;
END_VAR
```

#### Main.st
```iecst
PROGRAM _CYCLIC

	//Set FB parameter:
	MpAlarmXCore_0(
		Enable := TRUE,
		MpLink := ADR(gAlarmXCore));

	MpAlarmXListUI_0(
		MpLink := ADR(gAlarmXCore),
		Enable := TRUE,
		UIConnect := ADR(MpAlarmXListUIConnect));
	MpAlarmXHistory_0.MeasurementSystem := Test;
	MpAlarmXHistory_0(
		MpLink := ADR(gAlarmXHistory),
		Enable := TRUE,
		DeviceName := ADR('mappDir'),
		FileName := ADR('AlarmHistory_%Y_%m_%d_%H_%M_%S'),
		Language := ADR(gSetLanguage),
		MeasurementSystem := gSetUnit
	);

	//Show Alarm-Button in Visualization
	IF MpAlarmXCore_0.Active = TRUE THEN
		IF MpAlarmXCore_0.ActiveAlarms <> 0 OR MpAlarmXCore_0.PendingAlarms <> 0 THEN
			AlarmButton := 1;
			gCoffeeMainLogic.cmdAbort := TRUE;
			gCoffeeMainLogic.cmdClear := FALSE;
		ELSE
			AlarmButton := 0;
			gCoffeeMainLogic.cmdClear := TRUE;
			gCoffeeMainLogic.cmdAbort := FALSE;
		END_IF
	END_IF

	IF gCoffeeMainLogic.IdleState AND AlarmButton = 0 THEN
		ChangeStyleAlarmButton := 1;
	ELSE
		ChangeStyleAlarmButton := 0;
	END_IF

	IF MpAlarmXHistory_0.CommandDone = TRUE THEN
		MpAlarmXHistory_0.Export := FALSE;
	END_IF

	//Set Alarm-Video
	IF brsstrcmp(ADR(AlarmVideo), ADR("")) = 0 THEN
		AlarmInfo := FALSE;
	ELSE
		AlarmInfo := TRUE;
	END_IF

	FilterConfiguration;
	SortConfiguration;
	HistoryFilter;
	HistorySort;

END_PROGRAM
```

### Program Logical/Infrastructure/Recipe (IEC) - Recipe handling

#### Cyclic.ld - Cyclic code
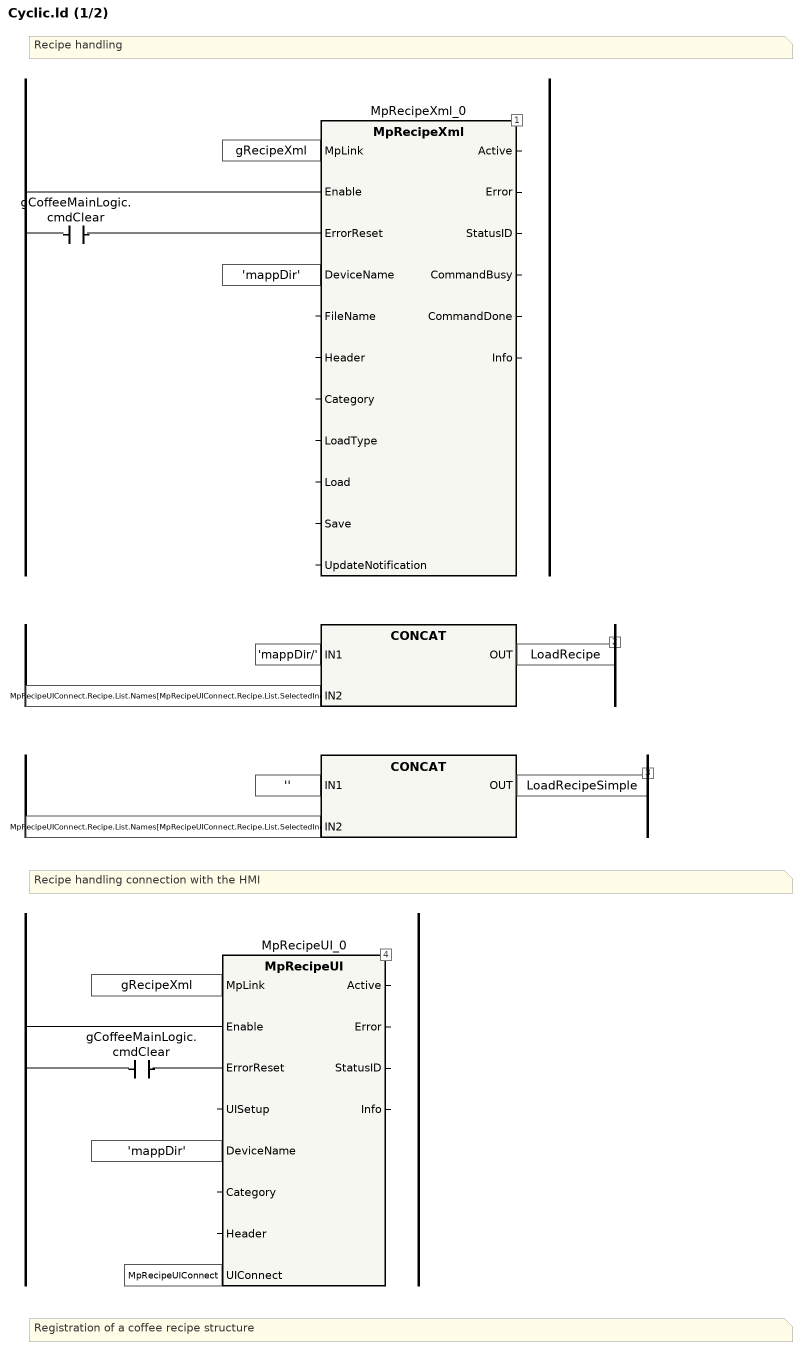
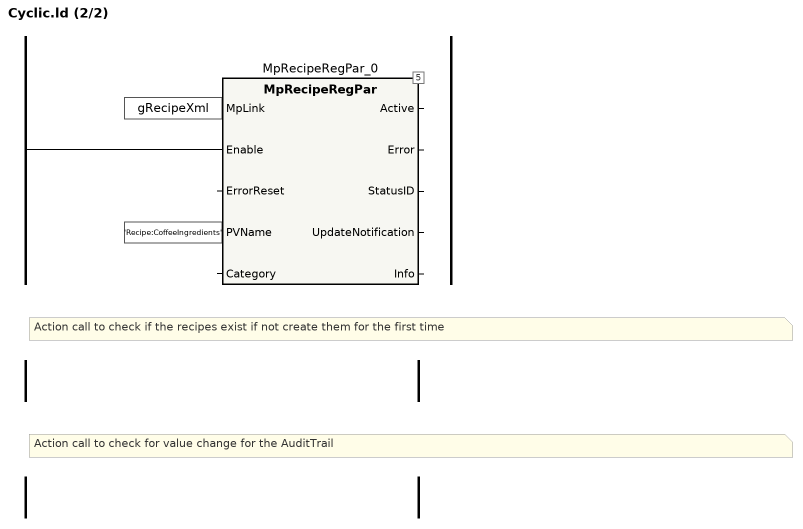
Diagram, in the editor's own instruction-list form stored in the file:
```il
PROGRAM _CYCLIC

VAR
	CreateRecipes_$$$$$$ : SFCActionType2;
	AuditTrail_$$$$$$ : SFCActionType2;
END_VAR

{NetworkNumber := 1}
(* Recipe handling *)
LD	gRecipeXml
ADR
ST	MpRecipeXml_0.MpLink
LD	TRUE
ST	MpRecipeXml_0.Enable
LD	gCoffeeMainLogic.cmdClear
ST	MpRecipeXml_0.ErrorReset
LD	'mappDir'
ADR
ST	MpRecipeXml_0.DeviceName
CAL	MpRecipeXml_0

{NetworkNumber := 2}
LD	'mappDir/'
CONCAT	MpRecipeUIConnect.Recipe.List.Names[MpRecipeUIConnect.Recipe.List.SelectedIndex]
ST	LoadRecipe

{NetworkNumber := 3}
LD	''
CONCAT	MpRecipeUIConnect.Recipe.List.Names[MpRecipeUIConnect.Recipe.List.SelectedIndex]
ST	LoadRecipeSimple

{NetworkNumber := 4}
(* Recipe handling connection with the HMI *)
LD	gRecipeXml
ADR
ST	MpRecipeUI_0.MpLink
LD	TRUE
ST	MpRecipeUI_0.Enable
LD	gCoffeeMainLogic.cmdClear
ST	MpRecipeUI_0.ErrorReset
LD	'mappDir'
ADR
ST	MpRecipeUI_0.DeviceName
LD	MpRecipeUIConnect
ADR
ST	MpRecipeUI_0.UIConnect
CAL	MpRecipeUI_0

{NetworkNumber := 5}
(* Registration of a coffee recipe structure *)
LD	gRecipeXml
ADR
ST	MpRecipeRegPar_0.MpLink
LD	TRUE
ST	MpRecipeRegPar_0.Enable
LD	'Recipe:CoffeeIngredients'
ADR
ST	MpRecipeRegPar_0.PVName
CAL	MpRecipeRegPar_0

{NetworkNumber := 6}
(* Action call to check if the recipes exist if not create them for the first time *)
LD	TRUE
S	CreateRecipes_$$$$$$.AC.N

{NetworkNumber := 7}
(* Action call to check for value change for the AuditTrail *)
LD	TRUE
S	AuditTrail_$$$$$$.AC.N

END_PROGRAM
```

#### Variables.var - Local variables
```iecst
VAR
	SaveRecipe : BOOL := FALSE;
	EditIngredients : CoffeeIngredientsType := (0);
	MpRecipeRegPar_0 : MpRecipeRegPar; (*Registration of the recipe structure variable*)
	TableConfiguration : STRING[80] := '{"specRows": [{"from":11, "to":20, "visible":false}]}';
	MpRecipeXml_0 : MpRecipeXml; (*Recipe Handling FUB*)
	MpRecipeUI_0 : MpRecipeUI := (UISetup:=(RecipeListSize:=11,RecipeListScrollWindow:=0,Confirmation:=(RecipeLoad:=0,RecipeSave:=0,RecipeCreate:=0,RecipeDelete:=TRUE))); (*MpRecipeUI Component*)
	RecipeCreateStep : RecipeCreateSteps := IDLE; (*Internal variable for recipe creating state machine*)
	MpRecipeUIConnect : MpRecipeUIConnectType := (Recipe:=(Filter:='*xml'),New:=(FileName:='newRecipe.xml')); (*MpRecipeUI connection datapoints*)
	CoffeeIngredients : CoffeeIngredientsType := (Milk:=100,Water:=150,Sugar:=30,Coffee:=60); (*Coffee machine recipe structure*)
END_VAR
(*Variables for AuditTrail*)
VAR
	_SelectedIndex : UINT := 0;
	LoadRecipe : STRING[80] := '0';
	DialogOpen : BOOL := 0;
	LoadRecipeSimple : STRING[255] := '0';
END_VAR
```

#### Types.typ - Local Variables
```iecst
TYPE
	RecipeCreateSteps :
		( (*Steps for creating recipes*)
		IDLE := 0, (*Idle State *)
		CREATE_1 := 10, (*Create coffee mappRegular*)
		DONE_1 := 11, (*mappRegular was created*)
		CREATE_2 := 20, (*Create coffee mappEspresso*)
		DONE_2 := 21, (*mappEspresso was created*)
		CREATE_3 := 30, (*Create coffee mappCappuccino*)
		DONE_3 := 31, (*mappCappuccino was created*)
		CREATE_4 := 40, (*Create coffee mappMilkCoffee*)
		DONE_4 := 41, (*mappMilkCoffee was created*)
		REFRESH := 42,
		LOAD := 43,
		ALL_DONE := 50 (*All recipes were created*)
		);
	CoffeeIngredientsType : 	STRUCT  (*Main ingredients structure*)
		Milk : INT; (*Amount of milk per cup*)
		Water : INT; (*Amount of water per cup*)
		Sugar : INT; (*Amount of sugar per cup*)
		Coffee : INT; (*Amount of coffee per cup*)
	END_STRUCT;
END_TYPE
```

#### CreateRecipes.st - Create recipes for the first time the project runs
```iecst
ACTION CreateRecipes:

	//Call TableConfiguration Variable
	TableConfiguration;

	// create default recipes in case they don't exist yet on the target
	// recipes are created by using the the MpRecipeXml instance interface

	CASE RecipeCreateStep OF
		IDLE:

			IF MpRecipeXml_0.Active = TRUE AND MpRecipeUI_0.Active = TRUE THEN

				// check for load error > triggers the default creation > if no error everything is ready to go
				IF (MpRecipeUIConnect.Recipe.List.Names[0] = '') THEN
					MpRecipeXml_0.Load 			:= FALSE;
					MpRecipeXml_0.ErrorReset 	:= TRUE;
					RecipeCreateStep 			:= CREATE_1;

				ELSIF (MpRecipeUIConnect.Recipe.List.Names[0] <> '' AND MpRecipeUI_0.Active = TRUE AND MpRecipeUIConnect.Status = mpRECIPE_UI_STATUS_IDLE) THEN
					MpRecipeUIConnect.Recipe.Load := TRUE;
				END_IF

				// reset the load command from the init when recipe was loaded successfully
				IF (MpRecipeUIConnect.Status = mpRECIPE_UI_STATUS_LOAD) AND (MpRecipeUIConnect.Recipe.Load = TRUE) THEN
					MpRecipeUIConnect.Recipe.Load			:= FALSE;
					RecipeCreateStep						:= ALL_DONE;
				END_IF

			END_IF

		CREATE_1:	// create the first recipe with default values, file name and a known picture index (Bitmap Group in the HMI)
			MpRecipeXml_0.ErrorReset 			:= FALSE;

			gCoffeeMainLogic.CreateFirstRecipe 	:= TRUE;
			CoffeeIngredients.Milk 				:= 0;
			CoffeeIngredients.Water 			:= 150;
			CoffeeIngredients.Sugar 			:= 0;
			CoffeeIngredients.Coffee 			:= 60;
			MpRecipeXml_0.FileName 				:= ADR('mappRegular.xml');
			MpRecipeXml_0.Save					:= TRUE;
			RecipeCreateStep 					:= DONE_1;

		DONE_1:	// when CommandDone GoTo next step
			IF(MpRecipeXml_0.CommandDone) THEN
				RecipeCreateStep 			:= CREATE_2;
				MpRecipeXml_0.Save			:= FALSE;
			END_IF;

		CREATE_2:	// create the next recipe with default values, file name and a known picture index (Bitmap Group in the HMI)

			CoffeeIngredients.Milk 				:= 0;
			CoffeeIngredients.Water 			:= 75;
			CoffeeIngredients.Sugar 			:= 0;
			CoffeeIngredients.Coffee 			:= 120;
			MpRecipeXml_0.FileName 				:= ADR('mappEspresso.xml');
			MpRecipeXml_0.Save					:= TRUE;
			RecipeCreateStep 					:= DONE_2;

		DONE_2:	// when CommandDone GoTo next step
			IF (MpRecipeXml_0.CommandDone) THEN
				RecipeCreateStep 			:= CREATE_3;
				MpRecipeXml_0.Save			:= FALSE;
			END_IF;

		CREATE_3:	// create the next recipe with default values, file name and a known picture index (Bitmap Group in the HMI)

			CoffeeIngredients.Milk 				:= 75;
			CoffeeIngredients.Water 			:= 75;
			CoffeeIngredients.Sugar 			:= 20;
			CoffeeIngredients.Coffee 			:= 120;
			MpRecipeXml_0.FileName 				:= ADR('mappCappuccino.xml');
			MpRecipeXml_0.Save					:= TRUE;
			RecipeCreateStep 					:= DONE_3;

		DONE_3:	// when CommandDone creating recipes is done
			IF(MpRecipeXml_0.CommandDone) THEN
				RecipeCreateStep 					:= CREATE_4;
				MpRecipeXml_0.Save					:= FALSE;
			END_IF;
		CREATE_4:	// create the next recipe with default values, file name and a known picture index (Bitmap Group in the HMI)

			CoffeeIngredients.Milk 				:= 100;
			CoffeeIngredients.Water 			:= 50;
			CoffeeIngredients.Sugar 			:= 0;
			CoffeeIngredients.Coffee 			:= 60;
			MpRecipeXml_0.FileName 				:= ADR('mappMilkCoffee.xml');
			MpRecipeXml_0.Save					:= TRUE;
			RecipeCreateStep 					:= REFRESH;

		REFRESH:	// refresh the recipe list to make sure all the recipes are shown

			IF(MpRecipeXml_0.CommandDone) THEN
				RecipeCreateStep 					:= LOAD;
				MpRecipeXml_0.Save					:= FALSE;
				MpRecipeUIConnect.Recipe.Refresh 	:= TRUE;
			END_IF;

		LOAD:	// load the first recipe to have a default recipe

			IF(MpRecipeUIConnect.Status = mpRECIPE_UI_STATUS_IDLE) AND MpRecipeUIConnect.Recipe.Refresh = FALSE THEN
				MpRecipeUIConnect.Recipe.Load 		:= TRUE;
				RecipeCreateStep 					:= DONE_4;
			END_IF

		DONE_4:	// if loading was successful the creation of the recipes is done

			IF(MpRecipeUIConnect.Status = mpRECIPE_UI_STATUS_IDLE)THEN
				RecipeCreateStep 					:= ALL_DONE;
				gCoffeeMainLogic.CreateFirstRecipe 	:= FALSE;
				MpRecipeUIConnect.Recipe.Refresh 	:= FALSE;
				MpRecipeUIConnect.Recipe.Load 		:= FALSE;
			END_IF;

	END_CASE;

	//Edit Recipe
	IF DialogOpen THEN

		EditIngredients.Milk 				:= CoffeeIngredients.Milk;
		EditIngredients.Water 				:= CoffeeIngredients.Water;
		EditIngredients.Sugar 				:= CoffeeIngredients.Sugar;
		EditIngredients.Coffee 				:= CoffeeIngredients.Coffee;
		DialogOpen 							:= FALSE;
	END_IF

	IF SaveRecipe THEN

		CoffeeIngredients.Milk 				:= EditIngredients.Milk;
		CoffeeIngredients.Water 			:= EditIngredients.Water;
		CoffeeIngredients.Sugar 			:= EditIngredients.Sugar;
		CoffeeIngredients.Coffee 			:= EditIngredients.Coffee;
	END_IF

END_ACTION
```

#### AuditTrail.st - Watch recipe variable for value change
```iecst
ACTION AuditTrail:

	//Load new recipe set recipe parameters
	IF MpRecipeUIConnect.Recipe.List.SelectedIndex <> _SelectedIndex AND MpRecipeUIConnect.Recipe.List.Names[0] <> '' AND MpRecipeUI_0.Active = TRUE AND MpRecipeUIConnect.Status = mpRECIPE_UI_STATUS_IDLE AND MpRecipeUIConnect.Recipe.Load = FALSE THEN
		_SelectedIndex := MpRecipeUIConnect.Recipe.List.SelectedIndex;
		MpRecipeUIConnect.Recipe.Load := TRUE;
	END_IF

	gCoffeeMainLogic.Refill[0] := CoffeeIngredients.Coffee ;
	gCoffeeMainLogic.Refill[1] := CoffeeIngredients.Milk ;
	gCoffeeMainLogic.Refill[2] := CoffeeIngredients.Sugar ;
	gCoffeeMainLogic.Refill[3] := CoffeeIngredients.Water ;

END_ACTION
```

### Program Logical/Infrastructure/File (IEC) - File manager

#### Cyclic.ld
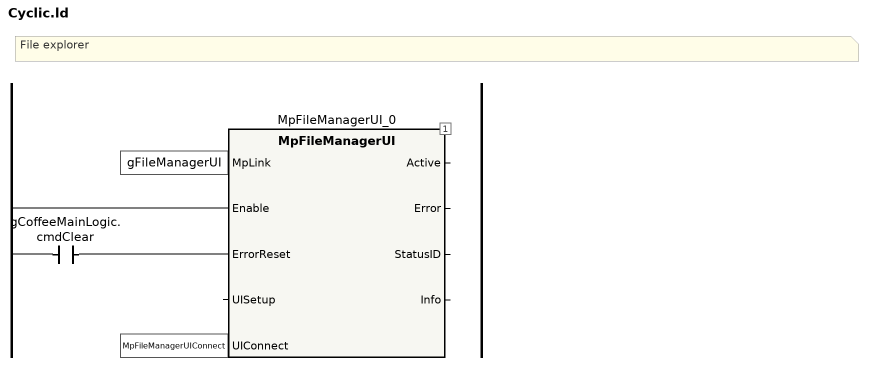
Diagram, in the editor's own instruction-list form stored in the file:
```il
PROGRAM _CYCLIC

{NetworkNumber := 1}
(* File explorer *)
LD	gFileManagerUI
ADR
ST	MpFileManagerUI_0.MpLink
LD	TRUE
ST	MpFileManagerUI_0.Enable
LD	gCoffeeMainLogic.cmdClear
ST	MpFileManagerUI_0.ErrorReset
LD	MpFileManagerUIConnect
ADR
ST	MpFileManagerUI_0.UIConnect
CAL	MpFileManagerUI_0

END_PROGRAM
```

#### Init.ld
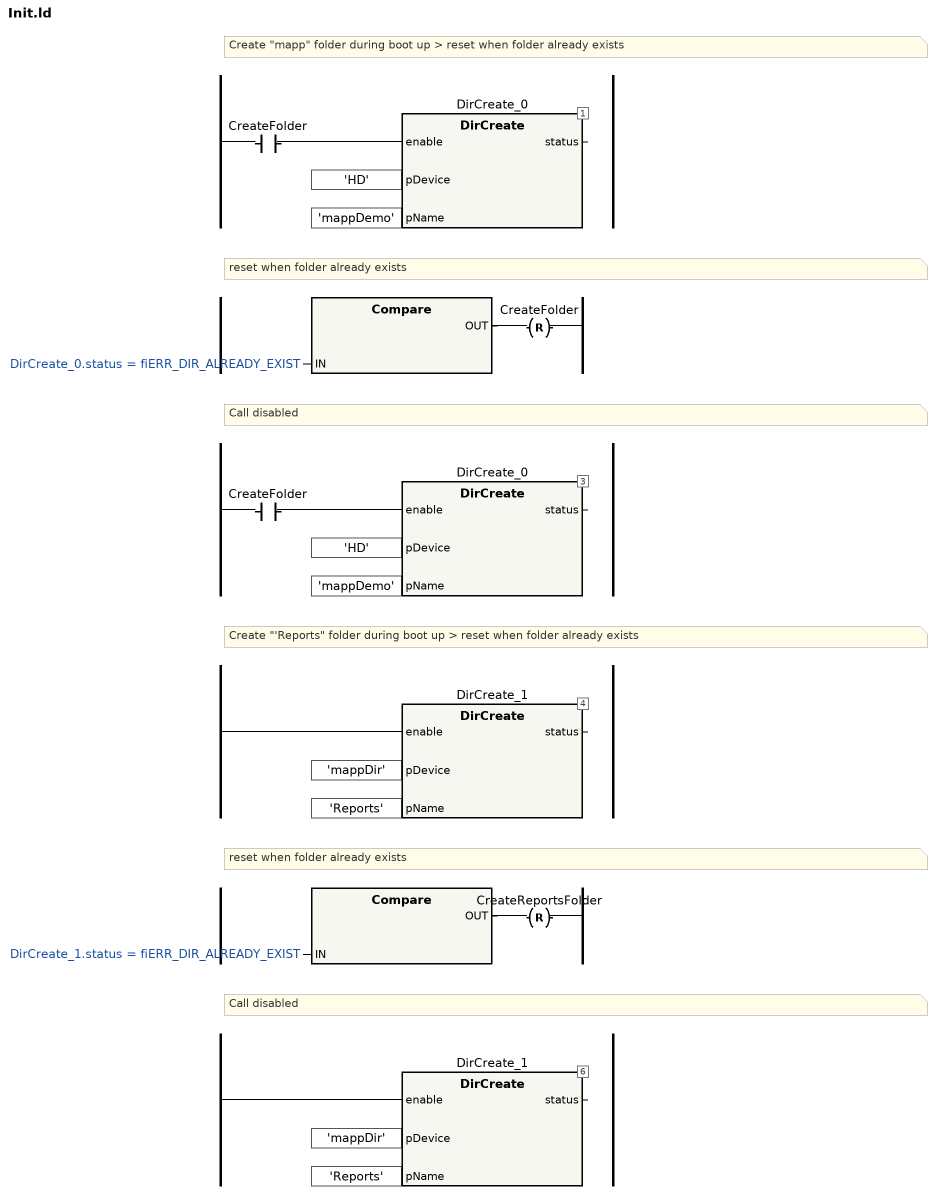
Diagram, in the editor's own instruction-list form stored in the file:
```il
PROGRAM _INIT

VAR
	zz$$$$_0_CompareBlock : ANY;
	zz$$$$_1_CompareBlock : ANY;
END_VAR

{NetworkNumber := 1}
(* Create "mapp" folder during boot up > reset when folder already exists *)
LD	CreateFolder
ST	DirCreate_0.enable
LD	'HD'
ADR
ST	DirCreate_0.pDevice
LD	'mappDemo'
ADR
ST	DirCreate_0.pName
CAL	DirCreate_0

{NetworkNumber := 2}
(* reset when folder already exists *)
Compare!	DirCreate_0.status = fiERR_DIR_ALREADY_EXIST
ST	zz$$$$_0_CompareBlock
R	CreateFolder

{NetworkNumber := 3}
(* Call disabled *)
LD	CreateFolder
ST	DirCreate_0.enable
LD	'HD'
ADR
ST	DirCreate_0.pDevice
LD	'mappDemo'
ADR
ST	DirCreate_0.pName
CAL	DirCreate_0

{NetworkNumber := 4}
(* Create "'Reports" folder during boot up > reset when folder already exists *)
LD	TRUE
ST	DirCreate_1.enable
LD	'mappDir'
ADR
ST	DirCreate_1.pDevice
LD	'Reports'
ADR
ST	DirCreate_1.pName
CAL	DirCreate_1

{NetworkNumber := 5}
(* reset when folder already exists *)
Compare!	DirCreate_1.status = fiERR_DIR_ALREADY_EXIST
ST	zz$$$$_1_CompareBlock
R	CreateReportsFolder

{NetworkNumber := 6}
(* Call disabled *)
LD	TRUE
ST	DirCreate_1.enable
LD	'mappDir'
ADR
ST	DirCreate_1.pDevice
LD	'Reports'
ADR
ST	DirCreate_1.pName
CAL	DirCreate_1

END_PROGRAM
```

### Program Logical/Infrastructure/Audit (IEC) - AuditTrail handling

#### Variables.var
```iecst
VAR
	MpAuditTrail_0 : MpAuditTrail; (*Parent component for change tracking*)
	MpAuditTrailUI_0 : MpAuditTrailUI := (UISetup:=(EventListSize:=20)); (*VC4 page connection  *)
	MpAuditTrailUIConnect : MpAuditTrailUIConnectType := (Filter:=(Dialog:=(From:=(Year:=1970,Month:=1,Day:=1,Hour:=00,Minute:=00),Until:=(Year:=1970,Month:=1,Day:=1,Hour:=00,Minute:=00)))); (*MpAuditTrailUI connection datapoints*)
	FilterConfiguration : STRING[2000] := '';
	SortConfiguraiton : STRING[2000] := '';
END_VAR
```

#### Cyclic.st
```iecst
PROGRAM _CYCLIC

	//Set FB parameters
	MpAuditTrail_0(
	MpLink := ADR(gAuditTrail),
	Enable := TRUE,
	DeviceName := ADR('mappDir'),
	ErrorReset := gCoffeeMainLogic.cmdClear,
	Language := ADR(gSetLanguage),
	FileName := ADR('Audit_%Y_%m_%d_%H_%M_%S'),
	MeasurementSystem := gSetUnit);

	MpAuditTrailUI_0(
	MpLink := ADR(gAuditTrail),
	Enable := TRUE,
	DeviceName := ADR('mappDir'),
	UIConnect := ADR(MpAuditTrailUIConnect),
	ErrorReset := gCoffeeMainLogic.cmdClear,
	Language := ADR(gSetLanguage),
	MeasurementSystem := gSetUnit);

	IF (MpAuditTrail_0.Export) AND (MpAuditTrail_0.CommandDone) THEN
		MpAuditTrail_0.Export := FALSE;
	END_IF

	IF MpAuditTrail_0.ArchiveAvailable THEN
		MpAuditTrail_0.ExportArchive := TRUE;
	ELSE
		MpAuditTrail_0.ExportArchive := FALSE;
	END_IF

	FilterConfiguration;
	SortConfiguraiton;

END_PROGRAM
```

### Program Logical/Infrastructure/Report (IEC) - Report handling

#### Variables.var
```iecst
VAR CONSTANT
	STR_FILE_DEVICE : STRING[80] := '/FileDevice:mappReport/';
END_VAR
VAR
	MpFileManagerUI_0 : MpFileManagerUI := (UISetup:=(FileListSize:=50));
	MpFileManagerUIConnect : MpFileManagerUIConnectType := (DeviceList:=(DeviceNames:=['mappReport',9('')]));
END_VAR
VAR CONSTANT
	REPORT_DEVICE : STRING[80] := 'mappReport'; (*Constant contains filedevice for save reports *)
	REPORT_NAME : STRING[80] := 'ReportCoffee'; (*Constant contains name of Report*)
END_VAR
VAR
	MpReportCore_0 : MpReportCore := (0); (*Core variable for MpReport*)
	DisplayFileName : ARRAY[0..49] OF STRING[255] := [50('')]; (*Displayed Files for mappView*)
	StrSelectedFile : STRING[256] := '0'; (*Gives the path of selected report to pdfViewer in mappView*)
	EnableGenerate : BOOL := TRUE; (*HMI control bit*)
	EnableDelete : BOOL := TRUE; (*HMI control bit*)
	i : USINT := 0; (*index for save filenames in a array*)
	DisplayFileNameIndex : USINT := 0; (*index of selected file for display in table in mappView*)
	DeleteReport : BOOL := 0; (*Start deleting a Report*)
	Refresh : BOOL := 0; (*strrt refresh process*)
	TON_0 : TON := (0); (*Timer to wait before refresh*)
END_VAR
```

#### Main.st
```iecst
PROGRAM _CYCLIC

	//Call FBs:
	MpReportCore_0(
		Enable := TRUE,
		MpLink := ADR(gReport),
		ReportID := ADR(REPORT_NAME),
		FileName := ADR('Report_%Y_%m_%d_%H_%M_%S'),
		DeviceName := ADR(REPORT_DEVICE),
		Language := ADR(gSetLanguage),
		MeasurementSystem := gSetUnit);
	MpFileManagerUI_0(MpLink := ADR(gReportFileManagerUI), UIConnect := ADR(MpFileManagerUIConnect), Enable := TRUE);

	//Call Action
	RefreshReport;

END_PROGRAM
```

#### RefreshReport.st
```iecst
ACTION RefreshReport:

	IF MpReportCore_0.Active = TRUE AND MpFileManagerUI_0.Active = TRUE THEN

		//Generate process
		IF MpReportCore_0.Generate = TRUE THEN

			IF MpReportCore_0.CommandDone = TRUE THEN

				MpReportCore_0.Generate := FALSE;
				Refresh := TRUE;
				EnableGenerate := FALSE;
			END_IF
		END_IF

		//Deleting process
		IF DeleteReport = TRUE THEN
			MpFileManagerUIConnect.File.Delete := TRUE;
			MpFileManagerUIConnect.MessageBox.Confirm := TRUE;
			DeleteReport := FALSE;
			Refresh := TRUE;
			EnableDelete := FALSE;
		END_IF

		//Refresh process
		IF Refresh = TRUE THEN
			TON_0(IN := TRUE, PT := T#2s);
			IF TON_0.Q = TRUE THEN
				Refresh := FALSE;
				TON_0(IN := FALSE, PT := T#2s);
				MpFileManagerUIConnect.File.Refresh := TRUE;
			END_IF
		END_IF

		//reset enable attribute for buttons
		IF Refresh = FALSE THEN
			EnableDelete := TRUE;
			EnableGenerate := TRUE;
		END_IF

		FOR i := 0 TO 49 DO
			// Save Filenames to a seperate array for display in Table
			DisplayFileName[i] := MpFileManagerUIConnect.File.List.Items[i].Name;
			IF DisplayFileNameIndex = i THEN
				// if selected set a index for display selected file in table
				MpFileManagerUIConnect.File.List.Items[i].IsSelected := TRUE;
			END_IF
		END_FOR

		// String for pdfViewer to display right report
		StrSelectedFile := CONCAT(STR_FILE_DEVICE, MpFileManagerUIConnect.File.List.Items[DisplayFileNameIndex].Name);

	END_IF

END_ACTION
```

### Program Logical/Infrastructure/IO (IEC) - Hardware handling

#### Variables.var
```iecst
VAR
	FileName : STRING[80] := ''; (*FileName of HWConfig file*)
	MpIOImport_0 : MpIOImport;
	ActiveConfiguration : STRING[80] := 'Configuration 1';
END_VAR
```

#### Main.st
```iecst
PROGRAM _INIT

END_PROGRAM
PROGRAM _CYCLIC

	ActiveConfiguration;

	//Set FB parameters
	MpIOImport_0(
		Enable := TRUE,
		MpLink := ADR(gIoConfig),
		DeviceName := ADR('mappIO'),
		FileName := ADR(FileName));

	//Reset Import command if import succeded
	IF MpIOImport_0.CommandDone = TRUE THEN
		MpIOImport_0.Import := FALSE;
	END_IF

END_PROGRAM
```

### Program Logical/Infrastructure/Sequence (IEC) - Sequencer handling
